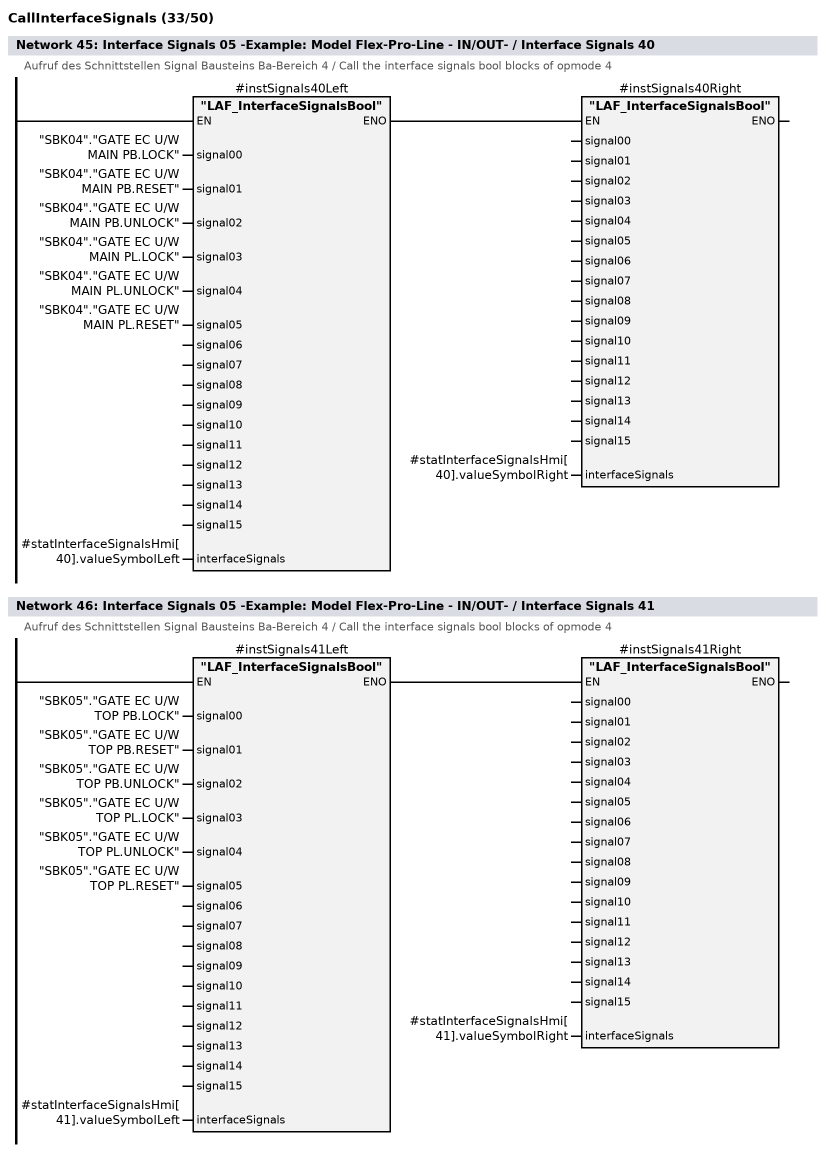
   RUNG wire#powerrail
      #instSignals40Left(signal00 := "SBK04"."GATE EC U/W MAIN PB.LOCK", signal01 := "SBK04"."GATE EC U/W MAIN PB.RESET", signal02 := "SBK04"."GATE EC U/W MAIN PB.UNLOCK", signal03 := "SBK04"."GATE EC U/W MAIN PL.LOCK", signal04 := "SBK04"."GATE EC U/W MAIN PL.UNLOCK", signal05 := "SBK04"."GATE EC U/W MAIN PL.RESET", signal06 :=, signal07 :=, signal08 :=, signal09 :=, signal10 :=, signal11 :=, signal12 :=, signal13 :=, signal14 :=, signal15 :=, interfaceSignals := #statInterfaceSignalsHmi[40].valueSymbolLeft)
      #instSignals40Right(signal00 :=, signal01 :=, signal02 :=, signal03 :=, signal04 :=, signal05 :=, signal06 :=, signal07 :=, signal08 :=, signal09 :=, signal10 :=, signal11 :=, signal12 :=, signal13 :=, signal14 :=, signal15 :=, interfaceSignals := #statInterfaceSignalsHmi[40].valueSymbolRight)
   END_RUNG
   // the same network as SCL:
   #instSignals40Left(signal00 := "SBK04"."GATE EC U/W MAIN PB.LOCK",   // "LAF_InterfaceSignalsBool"
                      signal01 := "SBK04"."GATE EC U/W MAIN PB.RESET",
                      signal02 := "SBK04"."GATE EC U/W MAIN PB.UNLOCK",
                      signal03 := "SBK04"."GATE EC U/W MAIN PL.LOCK",
                      signal04 := "SBK04"."GATE EC U/W MAIN PL.UNLOCK",
                      signal05 := "SBK04"."GATE EC U/W MAIN PL.RESET",
                      interfaceSignals := #statInterfaceSignalsHmi[40].valueSymbolLeft,
                      ENO => #_w1);
   IF #_w1 THEN
       #instSignals40Right(interfaceSignals := #statInterfaceSignalsHmi[40].valueSymbolRight);   // "LAF_InterfaceSignalsBool"
   END_IF;
END_REGION

REGION Network 46: Interface Signals 05 -Example: Model Flex-Pro-Line - IN/OUT- / Interface Signals 41
   // Aufruf des Schnittstellen Signal Bausteins Ba-Bereich 4 / Call the interface signals bool blocks of opmode 4
   RUNG wire#powerrail
      #instSignals41Left(signal00 := "SBK05"."GATE EC U/W TOP PB.LOCK", signal01 := "SBK05"."GATE EC U/W TOP PB.RESET", signal02 := "SBK05"."GATE EC U/W TOP PB.UNLOCK", signal03 := "SBK05"."GATE EC U/W TOP PL.LOCK", signal04 := "SBK05"."GATE EC U/W TOP PL.UNLOCK", signal05 := "SBK05"."GATE EC U/W TOP PL.RESET", signal06 :=, signal07 :=, signal08 :=, signal09 :=, signal10 :=, signal11 :=, signal12 :=, signal13 :=, signal14 :=, signal15 :=, interfaceSignals := #statInterfaceSignalsHmi[41].valueSymbolLeft)
      #instSignals41Right(signal00 :=, signal01 :=, signal02 :=, signal03 :=, signal04 :=, signal05 :=, signal06 :=, signal07 :=, signal08 :=, signal09 :=, signal10 :=, signal11 :=, signal12 :=, signal13 :=, signal14 :=, signal15 :=, interfaceSignals := #statInterfaceSignalsHmi[41].valueSymbolRight)
   END_RUNG
   // the same network as SCL:
   #instSignals41Left(signal00 := "SBK05"."GATE EC U/W TOP PB.LOCK",   // "LAF_InterfaceSignalsBool"
                      signal01 := "SBK05"."GATE EC U/W TOP PB.RESET",
                      signal02 := "SBK05"."GATE EC U/W TOP PB.UNLOCK",
                      signal03 := "SBK05"."GATE EC U/W TOP PL.LOCK",
                      signal04 := "SBK05"."GATE EC U/W TOP PL.UNLOCK",
                      signal05 := "SBK05"."GATE EC U/W TOP PL.RESET",
                      interfaceSignals := #statInterfaceSignalsHmi[41].valueSymbolLeft,
                      ENO => #_w1);
   IF #_w1 THEN
       #instSignals41Right(interfaceSignals := #statInterfaceSignalsHmi[41].valueSymbolRight);   // "LAF_InterfaceSignalsBool"
   END_IF;
END_REGION

REGION Network 47: Interface Signals 05 -Example: Model Flex-Pro-Line - IN/OUT- / Interface Signals 42
   // Aufruf des Schnittstellen Signal Bausteins Ba-Bereich 4 / Call the interface signals bool blocks of opmode 4
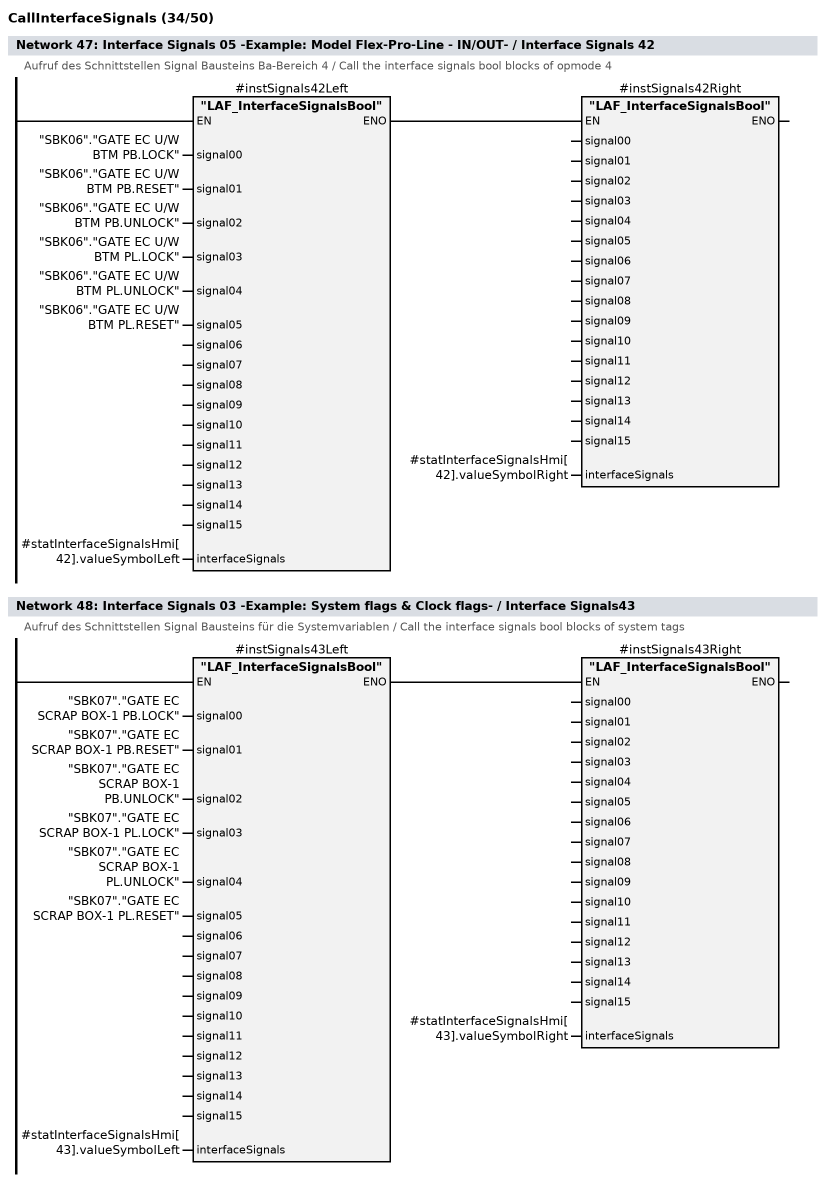
   RUNG wire#powerrail
      #instSignals42Left(signal00 := "SBK06"."GATE EC U/W BTM PB.LOCK", signal01 := "SBK06"."GATE EC U/W BTM PB.RESET", signal02 := "SBK06"."GATE EC U/W BTM PB.UNLOCK", signal03 := "SBK06"."GATE EC U/W BTM PL.LOCK", signal04 := "SBK06"."GATE EC U/W BTM PL.UNLOCK", signal05 := "SBK06"."GATE EC U/W BTM PL.RESET", signal06 :=, signal07 :=, signal08 :=, signal09 :=, signal10 :=, signal11 :=, signal12 :=, signal13 :=, signal14 :=, signal15 :=, interfaceSignals := #statInterfaceSignalsHmi[42].valueSymbolLeft)
      #instSignals42Right(signal00 :=, signal01 :=, signal02 :=, signal03 :=, signal04 :=, signal05 :=, signal06 :=, signal07 :=, signal08 :=, signal09 :=, signal10 :=, signal11 :=, signal12 :=, signal13 :=, signal14 :=, signal15 :=, interfaceSignals := #statInterfaceSignalsHmi[42].valueSymbolRight)
   END_RUNG
   // the same network as SCL:
   #instSignals42Left(signal00 := "SBK06"."GATE EC U/W BTM PB.LOCK",   // "LAF_InterfaceSignalsBool"
                      signal01 := "SBK06"."GATE EC U/W BTM PB.RESET",
                      signal02 := "SBK06"."GATE EC U/W BTM PB.UNLOCK",
                      signal03 := "SBK06"."GATE EC U/W BTM PL.LOCK",
                      signal04 := "SBK06"."GATE EC U/W BTM PL.UNLOCK",
                      signal05 := "SBK06"."GATE EC U/W BTM PL.RESET",
                      interfaceSignals := #statInterfaceSignalsHmi[42].valueSymbolLeft,
                      ENO => #_w1);
   IF #_w1 THEN
       #instSignals42Right(interfaceSignals := #statInterfaceSignalsHmi[42].valueSymbolRight);   // "LAF_InterfaceSignalsBool"
   END_IF;
END_REGION

REGION Network 48: Interface Signals 03 -Example: System flags & Clock flags- / Interface Signals43
   // Aufruf des Schnittstellen Signal Bausteins für die Systemvariablen / Call the interface signals bool blocks of system tags
   RUNG wire#powerrail
      #instSignals43Left(signal00 := "SBK07"."GATE EC SCRAP BOX-1 PB.LOCK", signal01 := "SBK07"."GATE EC SCRAP BOX-1 PB.RESET", signal02 := "SBK07"."GATE EC SCRAP BOX-1 PB.UNLOCK", signal03 := "SBK07"."GATE EC SCRAP BOX-1 PL.LOCK", signal04 := "SBK07"."GATE EC SCRAP BOX-1 PL.UNLOCK", signal05 := "SBK07"."GATE EC SCRAP BOX-1 PL.RESET", signal06 :=, signal07 :=, signal08 :=, signal09 :=, signal10 :=, signal11 :=, signal12 :=, signal13 :=, signal14 :=, signal15 :=, interfaceSignals := #statInterfaceSignalsHmi[43].valueSymbolLeft)
      #instSignals43Right(signal00 :=, signal01 :=, signal02 :=, signal03 :=, signal04 :=, signal05 :=, signal06 :=, signal07 :=, signal08 :=, signal09 :=, signal10 :=, signal11 :=, signal12 :=, signal13 :=, signal14 :=, signal15 :=, interfaceSignals := #statInterfaceSignalsHmi[43].valueSymbolRight)
   END_RUNG
   // the same network as SCL:
   #instSignals43Left(signal00 := "SBK07"."GATE EC SCRAP BOX-1 PB.LOCK",   // "LAF_InterfaceSignalsBool"
                      signal01 := "SBK07"."GATE EC SCRAP BOX-1 PB.RESET",
                      signal02 := "SBK07"."GATE EC SCRAP BOX-1 PB.UNLOCK",
                      signal03 := "SBK07"."GATE EC SCRAP BOX-1 PL.LOCK",
                      signal04 := "SBK07"."GATE EC SCRAP BOX-1 PL.UNLOCK",
                      signal05 := "SBK07"."GATE EC SCRAP BOX-1 PL.RESET",
                      interfaceSignals := #statInterfaceSignalsHmi[43].valueSymbolLeft,
                      ENO => #_w1);
   IF #_w1 THEN
       #instSignals43Right(interfaceSignals := #statInterfaceSignalsHmi[43].valueSymbolRight);   // "LAF_InterfaceSignalsBool"
   END_IF;
END_REGION

REGION Network 49: Interface Signals 04 -Example: Model Flex-Pro-Line - IN/OUT- / Interface Signals 44
   // Aufruf des Schnittstellen Signal Bausteins Ba-Bereich 4 / Call the interface signals bool blocks of opmode 4
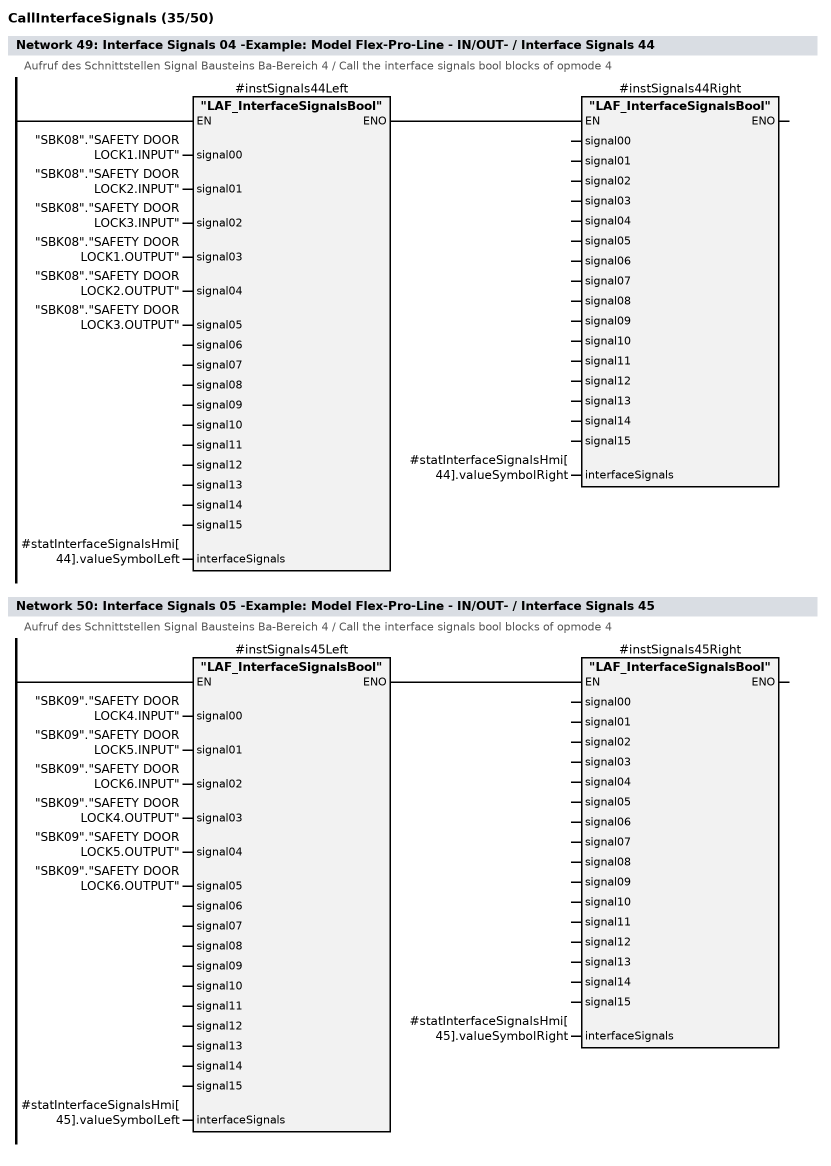
   RUNG wire#powerrail
      #instSignals44Left(signal00 := "SBK08"."SAFETY DOOR LOCK1.INPUT", signal01 := "SBK08"."SAFETY DOOR LOCK2.INPUT", signal02 := "SBK08"."SAFETY DOOR LOCK3.INPUT", signal03 := "SBK08"."SAFETY DOOR LOCK1.OUTPUT", signal04 := "SBK08"."SAFETY DOOR LOCK2.OUTPUT", signal05 := "SBK08"."SAFETY DOOR LOCK3.OUTPUT", signal06 :=, signal07 :=, signal08 :=, signal09 :=, signal10 :=, signal11 :=, signal12 :=, signal13 :=, signal14 :=, signal15 :=, interfaceSignals := #statInterfaceSignalsHmi[44].valueSymbolLeft)
      #instSignals44Right(signal00 :=, signal01 :=, signal02 :=, signal03 :=, signal04 :=, signal05 :=, signal06 :=, signal07 :=, signal08 :=, signal09 :=, signal10 :=, signal11 :=, signal12 :=, signal13 :=, signal14 :=, signal15 :=, interfaceSignals := #statInterfaceSignalsHmi[44].valueSymbolRight)
   END_RUNG
   // the same network as SCL:
   #instSignals44Left(signal00 := "SBK08"."SAFETY DOOR LOCK1.INPUT",   // "LAF_InterfaceSignalsBool"
                      signal01 := "SBK08"."SAFETY DOOR LOCK2.INPUT",
                      signal02 := "SBK08"."SAFETY DOOR LOCK3.INPUT",
                      signal03 := "SBK08"."SAFETY DOOR LOCK1.OUTPUT",
                      signal04 := "SBK08"."SAFETY DOOR LOCK2.OUTPUT",
                      signal05 := "SBK08"."SAFETY DOOR LOCK3.OUTPUT",
                      interfaceSignals := #statInterfaceSignalsHmi[44].valueSymbolLeft,
                      ENO => #_w1);
   IF #_w1 THEN
       #instSignals44Right(interfaceSignals := #statInterfaceSignalsHmi[44].valueSymbolRight);   // "LAF_InterfaceSignalsBool"
   END_IF;
END_REGION

REGION Network 50: Interface Signals 05 -Example: Model Flex-Pro-Line - IN/OUT- / Interface Signals 45
   // Aufruf des Schnittstellen Signal Bausteins Ba-Bereich 4 / Call the interface signals bool blocks of opmode 4
   RUNG wire#powerrail
      #instSignals45Left(signal00 := "SBK09"."SAFETY DOOR LOCK4.INPUT", signal01 := "SBK09"."SAFETY DOOR LOCK5.INPUT", signal02 := "SBK09"."SAFETY DOOR LOCK6.INPUT", signal03 := "SBK09"."SAFETY DOOR LOCK4.OUTPUT", signal04 := "SBK09"."SAFETY DOOR LOCK5.OUTPUT", signal05 := "SBK09"."SAFETY DOOR LOCK6.OUTPUT", signal06 :=, signal07 :=, signal08 :=, signal09 :=, signal10 :=, signal11 :=, signal12 :=, signal13 :=, signal14 :=, signal15 :=, interfaceSignals := #statInterfaceSignalsHmi[45].valueSymbolLeft)
      #instSignals45Right(signal00 :=, signal01 :=, signal02 :=, signal03 :=, signal04 :=, signal05 :=, signal06 :=, signal07 :=, signal08 :=, signal09 :=, signal10 :=, signal11 :=, signal12 :=, signal13 :=, signal14 :=, signal15 :=, interfaceSignals := #statInterfaceSignalsHmi[45].valueSymbolRight)
   END_RUNG
   // the same network as SCL:
   #instSignals45Left(signal00 := "SBK09"."SAFETY DOOR LOCK4.INPUT",   // "LAF_InterfaceSignalsBool"
                      signal01 := "SBK09"."SAFETY DOOR LOCK5.INPUT",
                      signal02 := "SBK09"."SAFETY DOOR LOCK6.INPUT",
                      signal03 := "SBK09"."SAFETY DOOR LOCK4.OUTPUT",
                      signal04 := "SBK09"."SAFETY DOOR LOCK5.OUTPUT",
                      signal05 := "SBK09"."SAFETY DOOR LOCK6.OUTPUT",
                      interfaceSignals := #statInterfaceSignalsHmi[45].valueSymbolLeft,
                      ENO => #_w1);
   IF #_w1 THEN
       #instSignals45Right(interfaceSignals := #statInterfaceSignalsHmi[45].valueSymbolRight);   // "LAF_InterfaceSignalsBool"
   END_IF;
END_REGION

REGION Network 51: Interface Signals 05 -Example: Model Flex-Pro-Line - IN/OUT- / Interface Signals 46
   // Aufruf des Schnittstellen Signal Bausteins Ba-Bereich 4 / Call the interface signals bool blocks of opmode 4
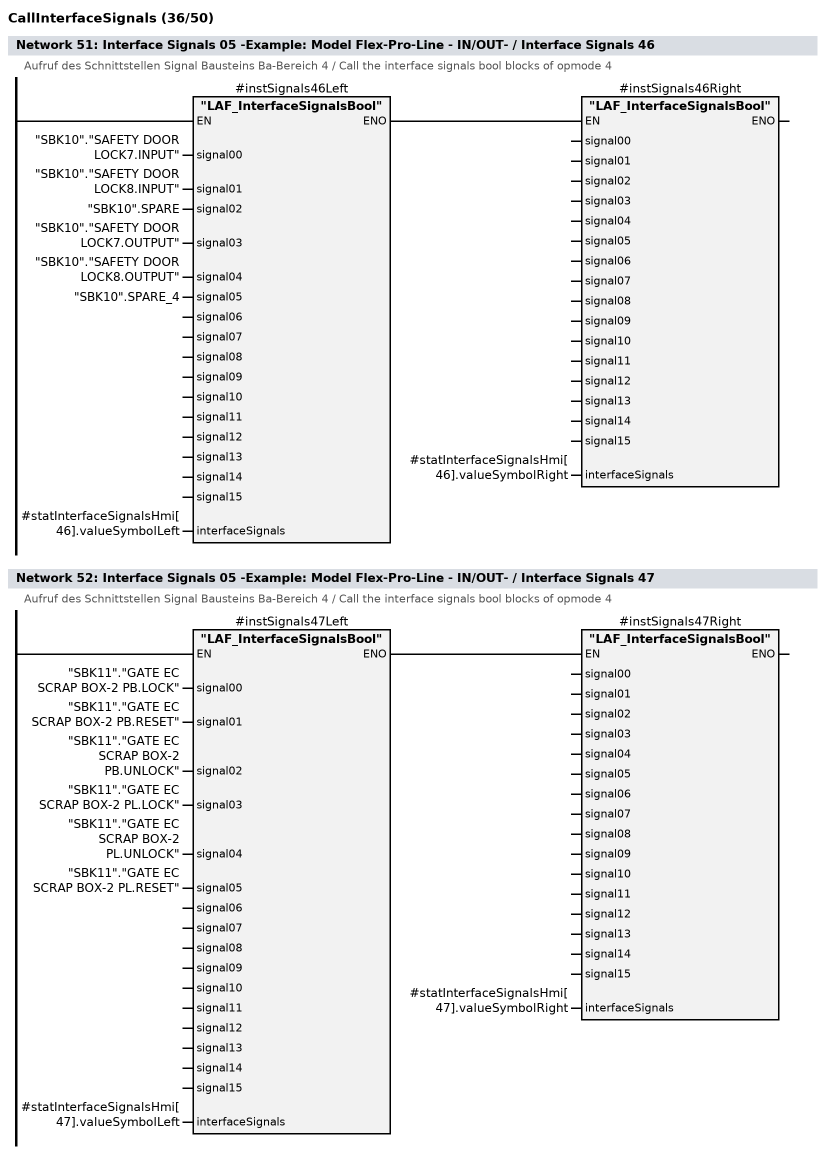
   RUNG wire#powerrail
      #instSignals46Left(signal00 := "SBK10"."SAFETY DOOR LOCK7.INPUT", signal01 := "SBK10"."SAFETY DOOR LOCK8.INPUT", signal02 := "SBK10".SPARE, signal03 := "SBK10"."SAFETY DOOR LOCK7.OUTPUT", signal04 := "SBK10"."SAFETY DOOR LOCK8.OUTPUT", signal05 := "SBK10".SPARE_4, signal06 :=, signal07 :=, signal08 :=, signal09 :=, signal10 :=, signal11 :=, signal12 :=, signal13 :=, signal14 :=, signal15 :=, interfaceSignals := #statInterfaceSignalsHmi[46].valueSymbolLeft)
      #instSignals46Right(signal00 :=, signal01 :=, signal02 :=, signal03 :=, signal04 :=, signal05 :=, signal06 :=, signal07 :=, signal08 :=, signal09 :=, signal10 :=, signal11 :=, signal12 :=, signal13 :=, signal14 :=, signal15 :=, interfaceSignals := #statInterfaceSignalsHmi[46].valueSymbolRight)
   END_RUNG
   // the same network as SCL:
   #instSignals46Left(signal00 := "SBK10"."SAFETY DOOR LOCK7.INPUT",   // "LAF_InterfaceSignalsBool"
                      signal01 := "SBK10"."SAFETY DOOR LOCK8.INPUT",
                      signal02 := "SBK10".SPARE,
                      signal03 := "SBK10"."SAFETY DOOR LOCK7.OUTPUT",
                      signal04 := "SBK10"."SAFETY DOOR LOCK8.OUTPUT",
                      signal05 := "SBK10".SPARE_4,
                      interfaceSignals := #statInterfaceSignalsHmi[46].valueSymbolLeft,
                      ENO => #_w1);
   IF #_w1 THEN
       #instSignals46Right(interfaceSignals := #statInterfaceSignalsHmi[46].valueSymbolRight);   // "LAF_InterfaceSignalsBool"
   END_IF;
END_REGION

REGION Network 52: Interface Signals 05 -Example: Model Flex-Pro-Line - IN/OUT- / Interface Signals 47
   // Aufruf des Schnittstellen Signal Bausteins Ba-Bereich 4 / Call the interface signals bool blocks of opmode 4
   RUNG wire#powerrail
      #instSignals47Left(signal00 := "SBK11"."GATE EC SCRAP BOX-2 PB.LOCK", signal01 := "SBK11"."GATE EC SCRAP BOX-2 PB.RESET", signal02 := "SBK11"."GATE EC SCRAP BOX-2 PB.UNLOCK", signal03 := "SBK11"."GATE EC SCRAP BOX-2 PL.LOCK", signal04 := "SBK11"."GATE EC SCRAP BOX-2 PL.UNLOCK", signal05 := "SBK11"."GATE EC SCRAP BOX-2 PL.RESET", signal06 :=, signal07 :=, signal08 :=, signal09 :=, signal10 :=, signal11 :=, signal12 :=, signal13 :=, signal14 :=, signal15 :=, interfaceSignals := #statInterfaceSignalsHmi[47].valueSymbolLeft)
      #instSignals47Right(signal00 :=, signal01 :=, signal02 :=, signal03 :=, signal04 :=, signal05 :=, signal06 :=, signal07 :=, signal08 :=, signal09 :=, signal10 :=, signal11 :=, signal12 :=, signal13 :=, signal14 :=, signal15 :=, interfaceSignals := #statInterfaceSignalsHmi[47].valueSymbolRight)
   END_RUNG
   // the same network as SCL:
   #instSignals47Left(signal00 := "SBK11"."GATE EC SCRAP BOX-2 PB.LOCK",   // "LAF_InterfaceSignalsBool"
                      signal01 := "SBK11"."GATE EC SCRAP BOX-2 PB.RESET",
                      signal02 := "SBK11"."GATE EC SCRAP BOX-2 PB.UNLOCK",
                      signal03 := "SBK11"."GATE EC SCRAP BOX-2 PL.LOCK",
                      signal04 := "SBK11"."GATE EC SCRAP BOX-2 PL.UNLOCK",
                      signal05 := "SBK11"."GATE EC SCRAP BOX-2 PL.RESET",
                      interfaceSignals := #statInterfaceSignalsHmi[47].valueSymbolLeft,
                      ENO => #_w1);
   IF #_w1 THEN
       #instSignals47Right(interfaceSignals := #statInterfaceSignalsHmi[47].valueSymbolRight);   // "LAF_InterfaceSignalsBool"
   END_IF;
END_REGION

REGION Network 53: Interface Signals 05 -Example: Model Flex-Pro-Line - IN/OUT- / Interface Signals 48
   // Aufruf des Schnittstellen Signal Bausteins Ba-Bereich 4 / Call the interface signals bool blocks of opmode 4
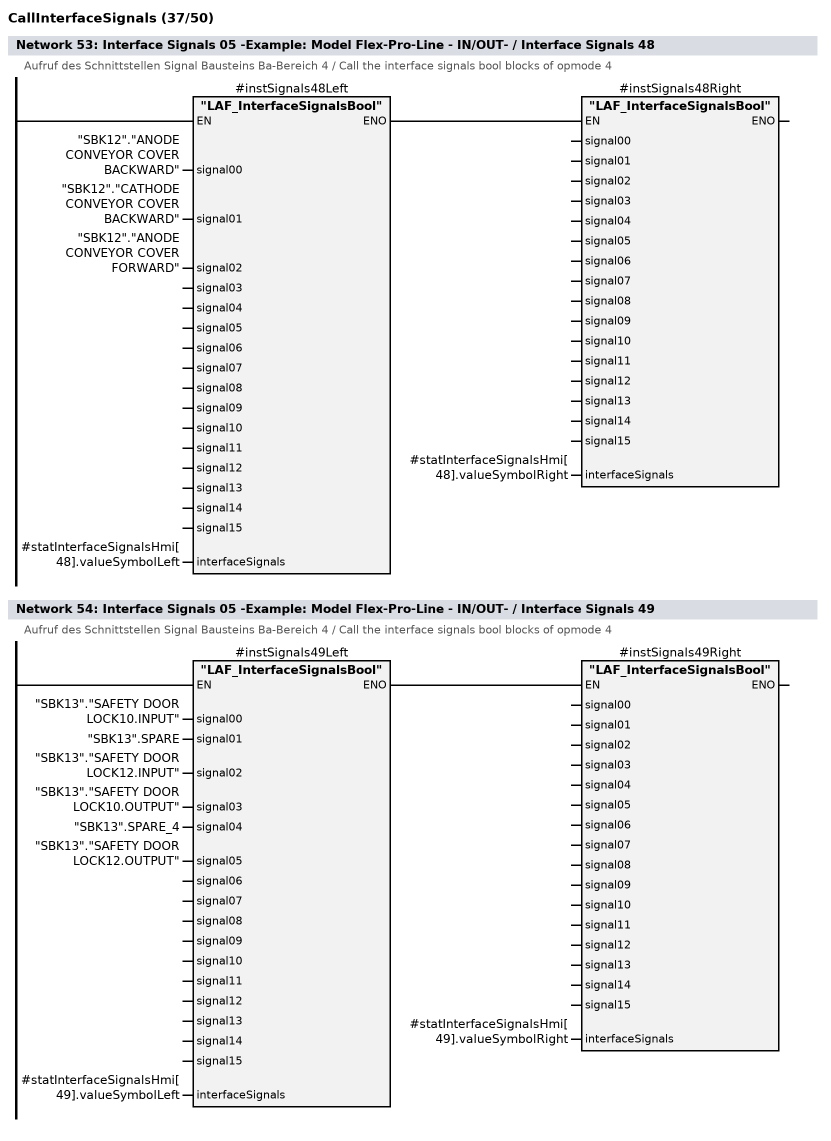
   RUNG wire#powerrail
      #instSignals48Left(signal00 := "SBK12"."ANODE CONVEYOR COVER BACKWARD", signal01 := "SBK12"."CATHODE CONVEYOR COVER BACKWARD", signal02 := "SBK12"."ANODE CONVEYOR COVER FORWARD", signal03 :=, signal04 :=, signal05 :=, signal06 :=, signal07 :=, signal08 :=, signal09 :=, signal10 :=, signal11 :=, signal12 :=, signal13 :=, signal14 :=, signal15 :=, interfaceSignals := #statInterfaceSignalsHmi[48].valueSymbolLeft)
      #instSignals48Right(signal00 :=, signal01 :=, signal02 :=, signal03 :=, signal04 :=, signal05 :=, signal06 :=, signal07 :=, signal08 :=, signal09 :=, signal10 :=, signal11 :=, signal12 :=, signal13 :=, signal14 :=, signal15 :=, interfaceSignals := #statInterfaceSignalsHmi[48].valueSymbolRight)
   END_RUNG
   // the same network as SCL:
   #instSignals48Left(signal00 := "SBK12"."ANODE CONVEYOR COVER BACKWARD",   // "LAF_InterfaceSignalsBool"
                      signal01 := "SBK12"."CATHODE CONVEYOR COVER BACKWARD",
                      signal02 := "SBK12"."ANODE CONVEYOR COVER FORWARD",
                      interfaceSignals := #statInterfaceSignalsHmi[48].valueSymbolLeft,
                      ENO => #_w1);
   IF #_w1 THEN
       #instSignals48Right(interfaceSignals := #statInterfaceSignalsHmi[48].valueSymbolRight);   // "LAF_InterfaceSignalsBool"
   END_IF;
END_REGION

REGION Network 54: Interface Signals 05 -Example: Model Flex-Pro-Line - IN/OUT- / Interface Signals 49
   // Aufruf des Schnittstellen Signal Bausteins Ba-Bereich 4 / Call the interface signals bool blocks of opmode 4
   RUNG wire#powerrail
      #instSignals49Left(signal00 := "SBK13"."SAFETY DOOR LOCK10.INPUT", signal01 := "SBK13".SPARE, signal02 := "SBK13"."SAFETY DOOR LOCK12.INPUT", signal03 := "SBK13"."SAFETY DOOR LOCK10.OUTPUT", signal04 := "SBK13".SPARE_4, signal05 := "SBK13"."SAFETY DOOR LOCK12.OUTPUT", signal06 :=, signal07 :=, signal08 :=, signal09 :=, signal10 :=, signal11 :=, signal12 :=, signal13 :=, signal14 :=, signal15 :=, interfaceSignals := #statInterfaceSignalsHmi[49].valueSymbolLeft)
      #instSignals49Right(signal00 :=, signal01 :=, signal02 :=, signal03 :=, signal04 :=, signal05 :=, signal06 :=, signal07 :=, signal08 :=, signal09 :=, signal10 :=, signal11 :=, signal12 :=, signal13 :=, signal14 :=, signal15 :=, interfaceSignals := #statInterfaceSignalsHmi[49].valueSymbolRight)
   END_RUNG
   // the same network as SCL:
   #instSignals49Left(signal00 := "SBK13"."SAFETY DOOR LOCK10.INPUT",   // "LAF_InterfaceSignalsBool"
                      signal01 := "SBK13".SPARE,
                      signal02 := "SBK13"."SAFETY DOOR LOCK12.INPUT",
                      signal03 := "SBK13"."SAFETY DOOR LOCK10.OUTPUT",
                      signal04 := "SBK13".SPARE_4,
                      signal05 := "SBK13"."SAFETY DOOR LOCK12.OUTPUT",
                      interfaceSignals := #statInterfaceSignalsHmi[49].valueSymbolLeft,
                      ENO => #_w1);
   IF #_w1 THEN
       #instSignals49Right(interfaceSignals := #statInterfaceSignalsHmi[49].valueSymbolRight);   // "LAF_InterfaceSignalsBool"
   END_IF;
END_REGION

REGION Network 55: Interface Signals 05 -Example: Model Flex-Pro-Line - IN/OUT- / Interface Signals 50
   // Aufruf des Schnittstellen Signal Bausteins Ba-Bereich 4 / Call the interface signals bool blocks of opmode 4
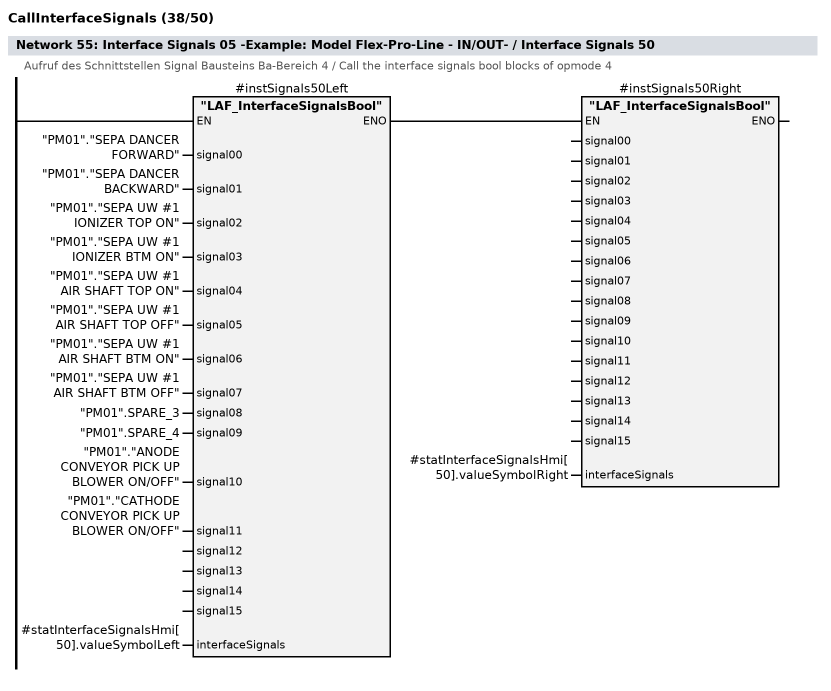
   RUNG wire#powerrail
      #instSignals50Left(signal00 := "PM01"."SEPA DANCER FORWARD", signal01 := "PM01"."SEPA DANCER BACKWARD", signal02 := "PM01"."SEPA UW #1 IONIZER TOP ON", signal03 := "PM01"."SEPA UW #1 IONIZER BTM ON", signal04 := "PM01"."SEPA UW #1 AIR SHAFT TOP ON", signal05 := "PM01"."SEPA UW #1 AIR SHAFT TOP OFF", signal06 := "PM01"."SEPA UW #1 AIR SHAFT BTM ON", signal07 := "PM01"."SEPA UW #1 AIR SHAFT BTM OFF", signal08 := "PM01".SPARE_3, signal09 := "PM01".SPARE_4, signal10 := "PM01"."ANODE CONVEYOR PICK UP BLOWER ON/OFF", signal11 := "PM01"."CATHODE CONVEYOR PICK UP BLOWER ON/OFF", signal12 :=, signal13 :=, signal14 :=, signal15 :=, interfaceSignals := #statInterfaceSignalsHmi[50].valueSymbolLeft)
      #instSignals50Right(signal00 :=, signal01 :=, signal02 :=, signal03 :=, signal04 :=, signal05 :=, signal06 :=, signal07 :=, signal08 :=, signal09 :=, signal10 :=, signal11 :=, signal12 :=, signal13 :=, signal14 :=, signal15 :=, interfaceSignals := #statInterfaceSignalsHmi[50].valueSymbolRight)
   END_RUNG
   // the same network as SCL:
   #instSignals50Left(signal00 := "PM01"."SEPA DANCER FORWARD",   // "LAF_InterfaceSignalsBool"
                      signal01 := "PM01"."SEPA DANCER BACKWARD",
                      signal02 := "PM01"."SEPA UW #1 IONIZER TOP ON",
                      signal03 := "PM01"."SEPA UW #1 IONIZER BTM ON",
                      signal04 := "PM01"."SEPA UW #1 AIR SHAFT TOP ON",
                      signal05 := "PM01"."SEPA UW #1 AIR SHAFT TOP OFF",
                      signal06 := "PM01"."SEPA UW #1 AIR SHAFT BTM ON",
                      signal07 := "PM01"."SEPA UW #1 AIR SHAFT BTM OFF",
                      signal08 := "PM01".SPARE_3,
                      signal09 := "PM01".SPARE_4,
                      signal10 := "PM01"."ANODE CONVEYOR PICK UP BLOWER ON/OFF",
                      signal11 := "PM01"."CATHODE CONVEYOR PICK UP BLOWER ON/OFF",
                      interfaceSignals := #statInterfaceSignalsHmi[50].valueSymbolLeft,
                      ENO => #_w1);
   IF #_w1 THEN
       #instSignals50Right(interfaceSignals := #statInterfaceSignalsHmi[50].valueSymbolRight);   // "LAF_InterfaceSignalsBool"
   END_IF;
END_REGION

REGION Network 56: Interface Signals 05 -Example: Model Flex-Pro-Line - IN/OUT- / Interface Signals 51
   // Aufruf des Schnittstellen Signal Bausteins Ba-Bereich 4 / Call the interface signals bool blocks of opmode 4
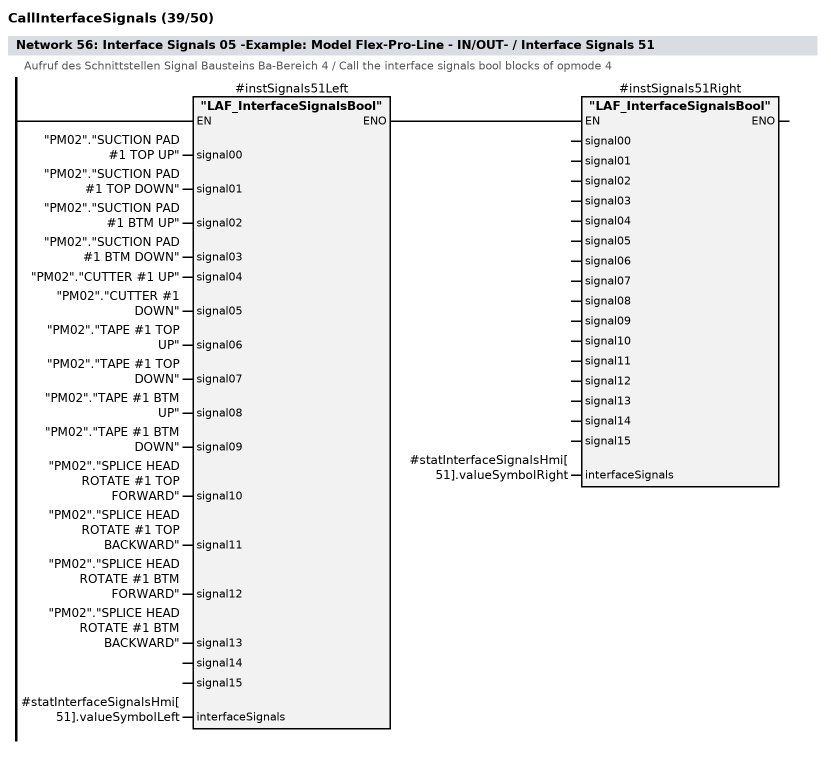
   RUNG wire#powerrail
      #instSignals51Left(signal00 := "PM02"."SUCTION PAD #1 TOP UP", signal01 := "PM02"."SUCTION PAD #1 TOP DOWN", signal02 := "PM02"."SUCTION PAD #1 BTM UP", signal03 := "PM02"."SUCTION PAD #1 BTM DOWN", signal04 := "PM02"."CUTTER #1 UP", signal05 := "PM02"."CUTTER #1 DOWN", signal06 := "PM02"."TAPE #1 TOP UP", signal07 := "PM02"."TAPE #1 TOP DOWN", signal08 := "PM02"."TAPE #1 BTM UP", signal09 := "PM02"."TAPE #1 BTM DOWN", signal10 := "PM02"."SPLICE HEAD ROTATE #1 TOP FORWARD", signal11 := "PM02"."SPLICE HEAD ROTATE #1 TOP BACKWARD", signal12 := "PM02"."SPLICE HEAD ROTATE #1 BTM FORWARD", signal13 := "PM02"."SPLICE HEAD ROTATE #1 BTM BACKWARD", signal14 :=, signal15 :=, interfaceSignals := #statInterfaceSignalsHmi[51].valueSymbolLeft)
      #instSignals51Right(signal00 :=, signal01 :=, signal02 :=, signal03 :=, signal04 :=, signal05 :=, signal06 :=, signal07 :=, signal08 :=, signal09 :=, signal10 :=, signal11 :=, signal12 :=, signal13 :=, signal14 :=, signal15 :=, interfaceSignals := #statInterfaceSignalsHmi[51].valueSymbolRight)
   END_RUNG
   // the same network as SCL:
   #instSignals51Left(signal00 := "PM02"."SUCTION PAD #1 TOP UP",   // "LAF_InterfaceSignalsBool"
                      signal01 := "PM02"."SUCTION PAD #1 TOP DOWN",
                      signal02 := "PM02"."SUCTION PAD #1 BTM UP",
                      signal03 := "PM02"."SUCTION PAD #1 BTM DOWN",
                      signal04 := "PM02"."CUTTER #1 UP",
                      signal05 := "PM02"."CUTTER #1 DOWN",
                      signal06 := "PM02"."TAPE #1 TOP UP",
                      signal07 := "PM02"."TAPE #1 TOP DOWN",
                      signal08 := "PM02"."TAPE #1 BTM UP",
                      signal09 := "PM02"."TAPE #1 BTM DOWN",
                      signal10 := "PM02"."SPLICE HEAD ROTATE #1 TOP FORWARD",
                      signal11 := "PM02"."SPLICE HEAD ROTATE #1 TOP BACKWARD",
                      signal12 := "PM02"."SPLICE HEAD ROTATE #1 BTM FORWARD",
                      signal13 := "PM02"."SPLICE HEAD ROTATE #1 BTM BACKWARD",
                      interfaceSignals := #statInterfaceSignalsHmi[51].valueSymbolLeft,
                      ENO => #_w1);
   IF #_w1 THEN
       #instSignals51Right(interfaceSignals := #statInterfaceSignalsHmi[51].valueSymbolRight);   // "LAF_InterfaceSignalsBool"
   END_IF;
END_REGION

REGION Network 57: Interface Signals 05 -Example: Model Flex-Pro-Line - IN/OUT- / Interface Signals 52
   // Aufruf des Schnittstellen Signal Bausteins Ba-Bereich 4 / Call the interface signals bool blocks of opmode 4
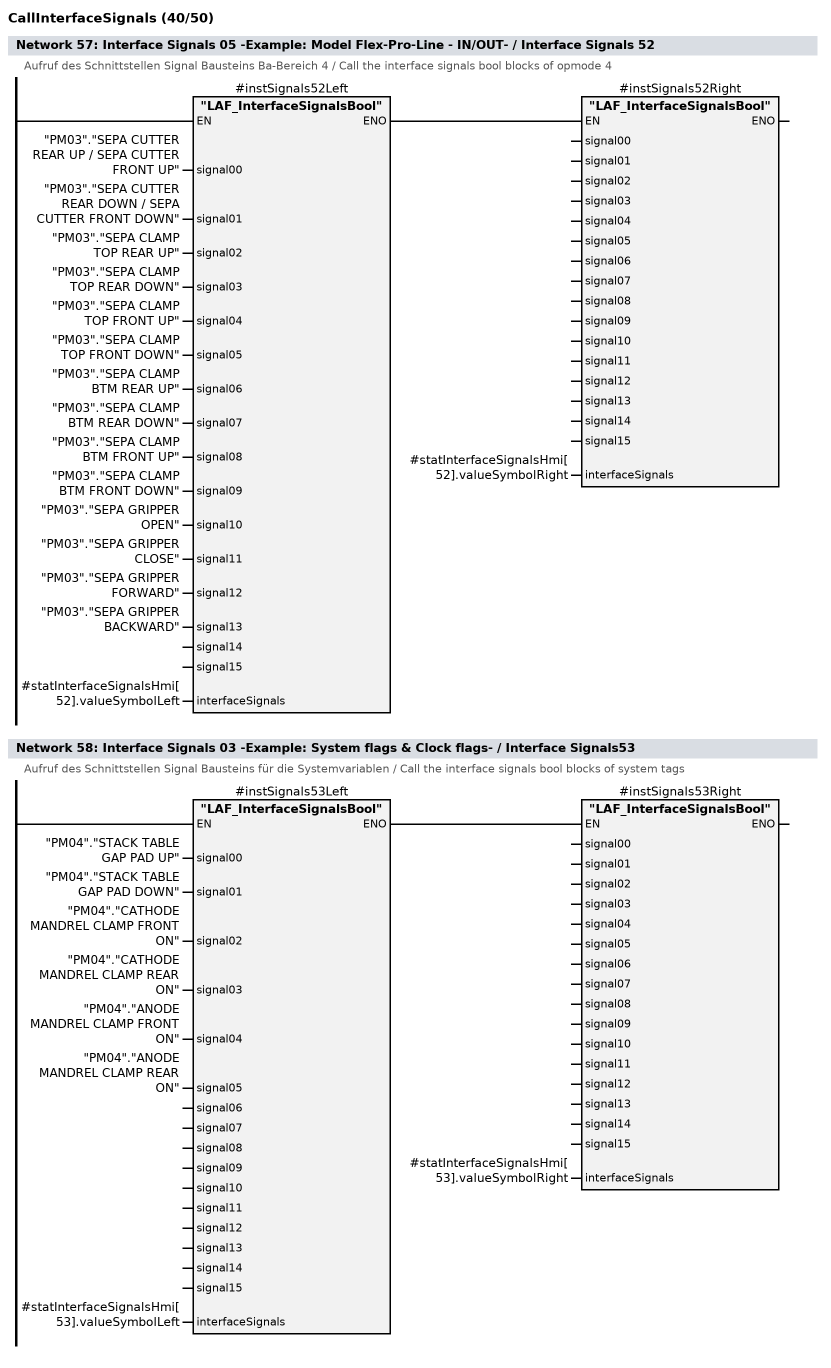
   RUNG wire#powerrail
      #instSignals52Left(signal00 := "PM03"."SEPA CUTTER REAR UP / SEPA CUTTER FRONT UP", signal01 := "PM03"."SEPA CUTTER REAR DOWN / SEPA CUTTER FRONT DOWN", signal02 := "PM03"."SEPA CLAMP TOP REAR UP", signal03 := "PM03"."SEPA CLAMP TOP REAR DOWN", signal04 := "PM03"."SEPA CLAMP TOP FRONT UP", signal05 := "PM03"."SEPA CLAMP TOP FRONT DOWN", signal06 := "PM03"."SEPA CLAMP BTM REAR UP", signal07 := "PM03"."SEPA CLAMP BTM REAR DOWN", signal08 := "PM03"."SEPA CLAMP BTM FRONT UP", signal09 := "PM03"."SEPA CLAMP BTM FRONT DOWN", signal10 := "PM03"."SEPA GRIPPER OPEN", signal11 := "PM03"."SEPA GRIPPER  CLOSE", signal12 := "PM03"."SEPA GRIPPER FORWARD", signal13 := "PM03"."SEPA GRIPPER BACKWARD", signal14 :=, signal15 :=, interfaceSignals := #statInterfaceSignalsHmi[52].valueSymbolLeft)
      #instSignals52Right(signal00 :=, signal01 :=, signal02 :=, signal03 :=, signal04 :=, signal05 :=, signal06 :=, signal07 :=, signal08 :=, signal09 :=, signal10 :=, signal11 :=, signal12 :=, signal13 :=, signal14 :=, signal15 :=, interfaceSignals := #statInterfaceSignalsHmi[52].valueSymbolRight)
   END_RUNG
   // the same network as SCL:
   #instSignals52Left(signal00 := "PM03"."SEPA CUTTER REAR UP / SEPA CUTTER FRONT UP",   // "LAF_InterfaceSignalsBool"
                      signal01 := "PM03"."SEPA CUTTER REAR DOWN / SEPA CUTTER FRONT DOWN",
                      signal02 := "PM03"."SEPA CLAMP TOP REAR UP",
                      signal03 := "PM03"."SEPA CLAMP TOP REAR DOWN",
                      signal04 := "PM03"."SEPA CLAMP TOP FRONT UP",
                      signal05 := "PM03"."SEPA CLAMP TOP FRONT DOWN",
                      signal06 := "PM03"."SEPA CLAMP BTM REAR UP",
                      signal07 := "PM03"."SEPA CLAMP BTM REAR DOWN",
                      signal08 := "PM03"."SEPA CLAMP BTM FRONT UP",
                      signal09 := "PM03"."SEPA CLAMP BTM FRONT DOWN",
                      signal10 := "PM03"."SEPA GRIPPER OPEN",
                      signal11 := "PM03"."SEPA GRIPPER  CLOSE",
                      signal12 := "PM03"."SEPA GRIPPER FORWARD",
                      signal13 := "PM03"."SEPA GRIPPER BACKWARD",
                      interfaceSignals := #statInterfaceSignalsHmi[52].valueSymbolLeft,
                      ENO => #_w1);
   IF #_w1 THEN
       #instSignals52Right(interfaceSignals := #statInterfaceSignalsHmi[52].valueSymbolRight);   // "LAF_InterfaceSignalsBool"
   END_IF;
END_REGION

REGION Network 58: Interface Signals 03 -Example: System flags & Clock flags- / Interface Signals53
   // Aufruf des Schnittstellen Signal Bausteins für die Systemvariablen / Call the interface signals bool blocks of system tags
   RUNG wire#powerrail
      #instSignals53Left(signal00 := "PM04"."STACK TABLE GAP PAD UP", signal01 := "PM04"."STACK TABLE GAP PAD DOWN", signal02 := "PM04"."CATHODE MANDREL CLAMP FRONT ON", signal03 := "PM04"."CATHODE MANDREL CLAMP REAR ON", signal04 := "PM04"."ANODE MANDREL CLAMP FRONT ON", signal05 := "PM04"."ANODE MANDREL CLAMP REAR ON", signal06 :=, signal07 :=, signal08 :=, signal09 :=, signal10 :=, signal11 :=, signal12 :=, signal13 :=, signal14 :=, signal15 :=, interfaceSignals := #statInterfaceSignalsHmi[53].valueSymbolLeft)
      #instSignals53Right(signal00 :=, signal01 :=, signal02 :=, signal03 :=, signal04 :=, signal05 :=, signal06 :=, signal07 :=, signal08 :=, signal09 :=, signal10 :=, signal11 :=, signal12 :=, signal13 :=, signal14 :=, signal15 :=, interfaceSignals := #statInterfaceSignalsHmi[53].valueSymbolRight)
   END_RUNG
   // the same network as SCL:
   #instSignals53Left(signal00 := "PM04"."STACK TABLE GAP PAD UP",   // "LAF_InterfaceSignalsBool"
                      signal01 := "PM04"."STACK TABLE GAP PAD DOWN",
                      signal02 := "PM04"."CATHODE MANDREL CLAMP FRONT ON",
                      signal03 := "PM04"."CATHODE MANDREL CLAMP REAR ON",
                      signal04 := "PM04"."ANODE MANDREL CLAMP FRONT ON",
                      signal05 := "PM04"."ANODE MANDREL CLAMP REAR ON",
                      interfaceSignals := #statInterfaceSignalsHmi[53].valueSymbolLeft,
                      ENO => #_w1);
   IF #_w1 THEN
       #instSignals53Right(interfaceSignals := #statInterfaceSignalsHmi[53].valueSymbolRight);   // "LAF_InterfaceSignalsBool"
   END_IF;
END_REGION

REGION Network 59: Interface Signals 04 -Example: Model Flex-Pro-Line - IN/OUT- / Interface Signals 54
   // Aufruf des Schnittstellen Signal Bausteins Ba-Bereich 4 / Call the interface signals bool blocks of opmode 4
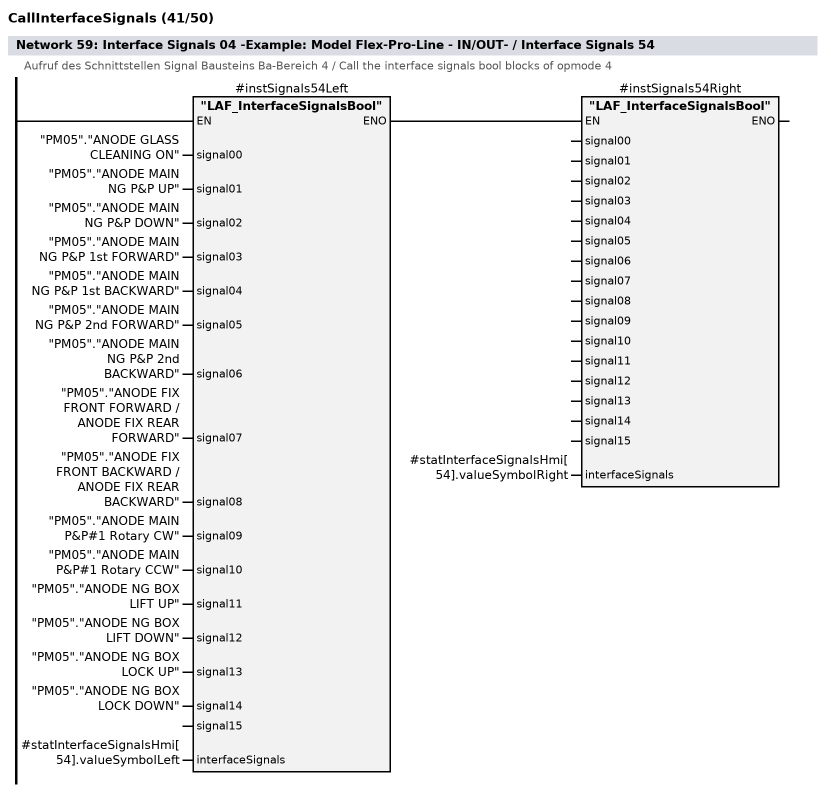
   RUNG wire#powerrail
      #instSignals54Left(signal00 := "PM05"."ANODE GLASS CLEANING ON", signal01 := "PM05"."ANODE MAIN NG P&P UP", signal02 := "PM05"."ANODE MAIN NG P&P DOWN", signal03 := "PM05"."ANODE MAIN NG P&P 1st FORWARD", signal04 := "PM05"."ANODE MAIN NG P&P 1st BACKWARD", signal05 := "PM05"."ANODE MAIN NG P&P 2nd FORWARD", signal06 := "PM05"."ANODE MAIN NG P&P 2nd BACKWARD", signal07 := "PM05"."ANODE FIX FRONT FORWARD / ANODE FIX REAR FORWARD", signal08 := "PM05"."ANODE FIX FRONT BACKWARD / ANODE FIX REAR BACKWARD", signal09 := "PM05"."ANODE MAIN P&P#1 Rotary CW", signal10 := "PM05"."ANODE MAIN P&P#1 Rotary CCW", signal11 := "PM05"."ANODE NG BOX LIFT UP", signal12 := "PM05"."ANODE NG BOX LIFT DOWN", signal13 := "PM05"."ANODE NG BOX LOCK UP", signal14 := "PM05"."ANODE NG BOX LOCK DOWN", signal15 :=, interfaceSignals := #statInterfaceSignalsHmi[54].valueSymbolLeft)
      #instSignals54Right(signal00 :=, signal01 :=, signal02 :=, signal03 :=, signal04 :=, signal05 :=, signal06 :=, signal07 :=, signal08 :=, signal09 :=, signal10 :=, signal11 :=, signal12 :=, signal13 :=, signal14 :=, signal15 :=, interfaceSignals := #statInterfaceSignalsHmi[54].valueSymbolRight)
   END_RUNG
   // the same network as SCL:
   #instSignals54Left(signal00 := "PM05"."ANODE GLASS CLEANING ON",   // "LAF_InterfaceSignalsBool"
                      signal01 := "PM05"."ANODE MAIN NG P&P UP",
                      signal02 := "PM05"."ANODE MAIN NG P&P DOWN",
                      signal03 := "PM05"."ANODE MAIN NG P&P 1st FORWARD",
                      signal04 := "PM05"."ANODE MAIN NG P&P 1st BACKWARD",
                      signal05 := "PM05"."ANODE MAIN NG P&P 2nd FORWARD",
                      signal06 := "PM05"."ANODE MAIN NG P&P 2nd BACKWARD",
                      signal07 := "PM05"."ANODE FIX FRONT FORWARD / ANODE FIX REAR FORWARD",
                      signal08 := "PM05"."ANODE FIX FRONT BACKWARD / ANODE FIX REAR BACKWARD",
                      signal09 := "PM05"."ANODE MAIN P&P#1 Rotary CW",
                      signal10 := "PM05"."ANODE MAIN P&P#1 Rotary CCW",
                      signal11 := "PM05"."ANODE NG BOX LIFT UP",
                      signal12 := "PM05"."ANODE NG BOX LIFT DOWN",
                      signal13 := "PM05"."ANODE NG BOX LOCK UP",
                      signal14 := "PM05"."ANODE NG BOX LOCK DOWN",
                      interfaceSignals := #statInterfaceSignalsHmi[54].valueSymbolLeft,
                      ENO => #_w1);
   IF #_w1 THEN
       #instSignals54Right(interfaceSignals := #statInterfaceSignalsHmi[54].valueSymbolRight);   // "LAF_InterfaceSignalsBool"
   END_IF;
END_REGION

REGION Network 60: Interface Signals 05 -Example: Model Flex-Pro-Line - IN/OUT- / Interface Signals 55
   // Aufruf des Schnittstellen Signal Bausteins Ba-Bereich 4 / Call the interface signals bool blocks of opmode 4
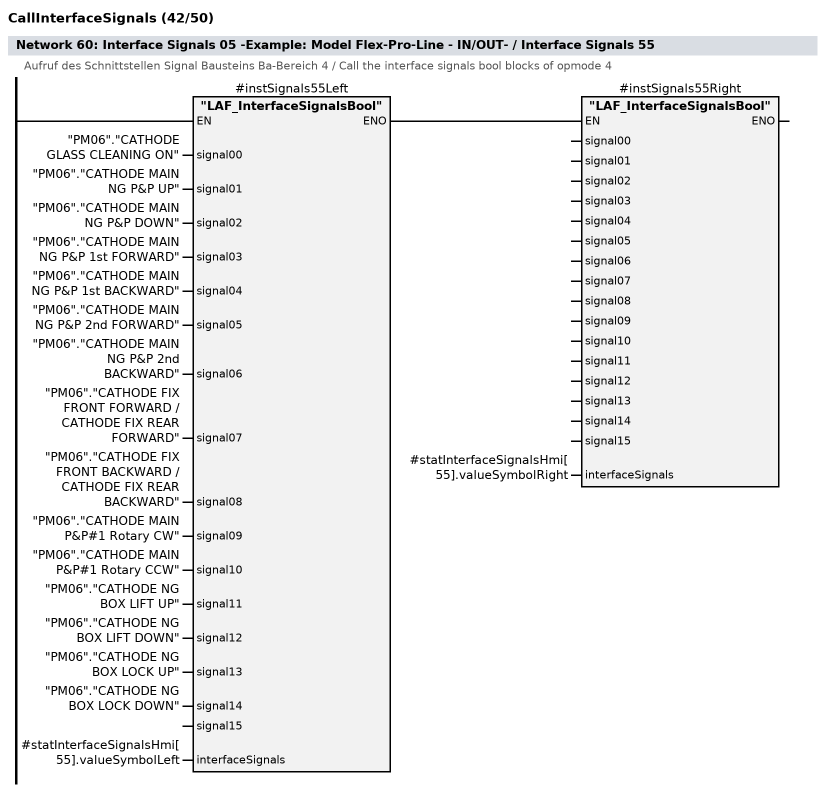
   RUNG wire#powerrail
      #instSignals55Left(signal00 := "PM06"."CATHODE GLASS CLEANING ON", signal01 := "PM06"."CATHODE MAIN NG P&P UP", signal02 := "PM06"."CATHODE MAIN NG P&P DOWN", signal03 := "PM06"."CATHODE MAIN NG P&P 1st FORWARD", signal04 := "PM06"."CATHODE MAIN NG P&P 1st BACKWARD", signal05 := "PM06"."CATHODE MAIN NG P&P 2nd FORWARD", signal06 := "PM06"."CATHODE MAIN NG P&P 2nd BACKWARD", signal07 := "PM06"."CATHODE FIX FRONT FORWARD / CATHODE FIX REAR FORWARD", signal08 := "PM06"."CATHODE FIX FRONT BACKWARD / CATHODE FIX REAR BACKWARD", signal09 := "PM06"."CATHODE MAIN P&P#1 Rotary CW", signal10 := "PM06"."CATHODE MAIN P&P#1 Rotary CCW", signal11 := "PM06"."CATHODE NG BOX LIFT UP", signal12 := "PM06"."CATHODE NG BOX LIFT DOWN", signal13 := "PM06"."CATHODE NG BOX LOCK UP", signal14 := "PM06"."CATHODE NG BOX LOCK DOWN", signal15 :=, interfaceSignals := #statInterfaceSignalsHmi[55].valueSymbolLeft)
      #instSignals55Right(signal00 :=, signal01 :=, signal02 :=, signal03 :=, signal04 :=, signal05 :=, signal06 :=, signal07 :=, signal08 :=, signal09 :=, signal10 :=, signal11 :=, signal12 :=, signal13 :=, signal14 :=, signal15 :=, interfaceSignals := #statInterfaceSignalsHmi[55].valueSymbolRight)
   END_RUNG
   // the same network as SCL:
   #instSignals55Left(signal00 := "PM06"."CATHODE GLASS CLEANING ON",   // "LAF_InterfaceSignalsBool"
                      signal01 := "PM06"."CATHODE MAIN NG P&P UP",
                      signal02 := "PM06"."CATHODE MAIN NG P&P DOWN",
                      signal03 := "PM06"."CATHODE MAIN NG P&P 1st FORWARD",
                      signal04 := "PM06"."CATHODE MAIN NG P&P 1st BACKWARD",
                      signal05 := "PM06"."CATHODE MAIN NG P&P 2nd FORWARD",
                      signal06 := "PM06"."CATHODE MAIN NG P&P 2nd BACKWARD",
                      signal07 := "PM06"."CATHODE FIX FRONT FORWARD / CATHODE FIX REAR FORWARD",
                      signal08 := "PM06"."CATHODE FIX FRONT BACKWARD / CATHODE FIX REAR BACKWARD",
                      signal09 := "PM06"."CATHODE MAIN P&P#1 Rotary CW",
                      signal10 := "PM06"."CATHODE MAIN P&P#1 Rotary CCW",
                      signal11 := "PM06"."CATHODE NG BOX LIFT UP",
                      signal12 := "PM06"."CATHODE NG BOX LIFT DOWN",
                      signal13 := "PM06"."CATHODE NG BOX LOCK UP",
                      signal14 := "PM06"."CATHODE NG BOX LOCK DOWN",
                      interfaceSignals := #statInterfaceSignalsHmi[55].valueSymbolLeft,
                      ENO => #_w1);
   IF #_w1 THEN
       #instSignals55Right(interfaceSignals := #statInterfaceSignalsHmi[55].valueSymbolRight);   // "LAF_InterfaceSignalsBool"
   END_IF;
END_REGION

REGION Network 61: Interface Signals 05 -Example: Model Flex-Pro-Line - IN/OUT- / Interface Signals 56
   // Aufruf des Schnittstellen Signal Bausteins Ba-Bereich 4 / Call the interface signals bool blocks of opmode 4
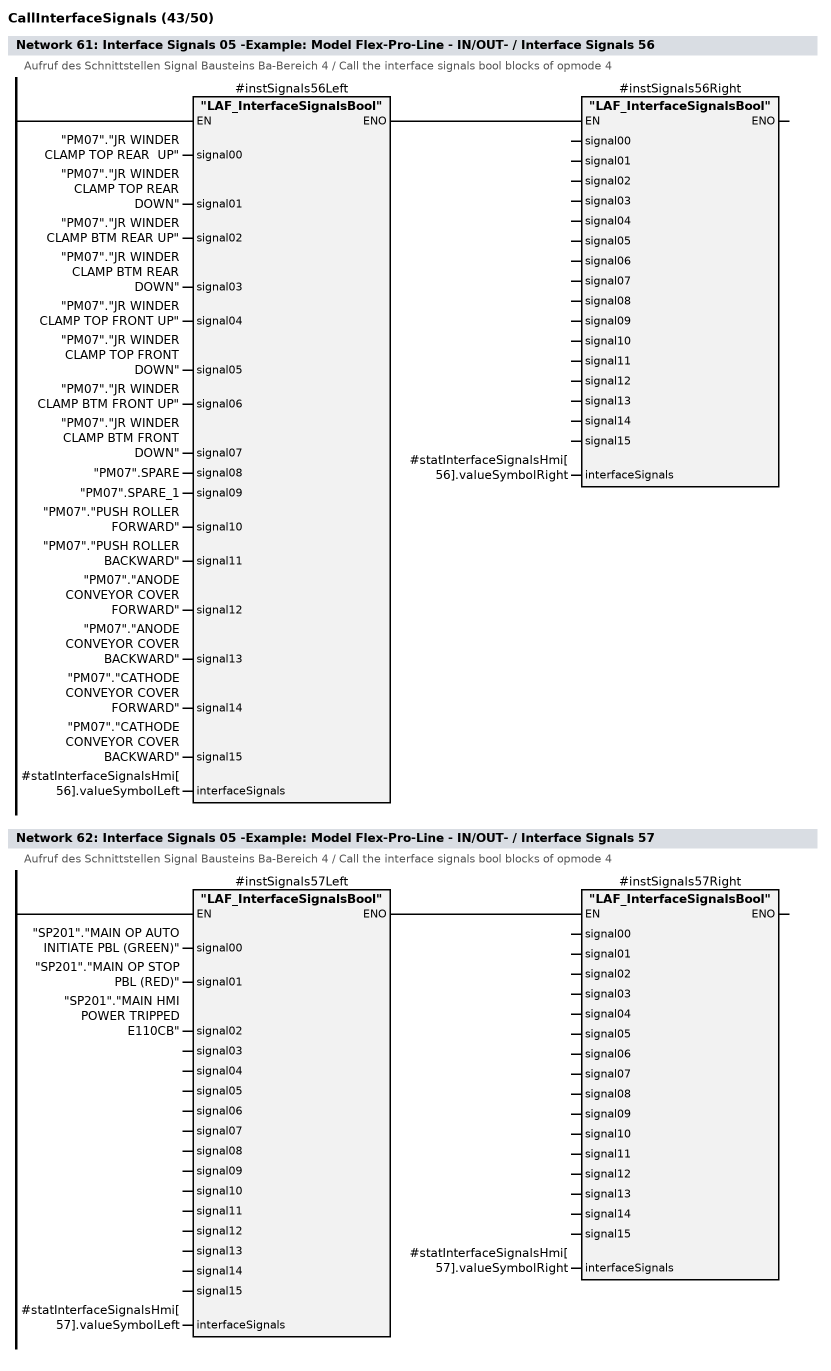
   RUNG wire#powerrail
      #instSignals56Left(signal00 := "PM07"."JR WINDER CLAMP TOP REAR  UP", signal01 := "PM07"."JR WINDER CLAMP TOP REAR  DOWN", signal02 := "PM07"."JR WINDER CLAMP BTM REAR UP", signal03 := "PM07"."JR WINDER CLAMP BTM REAR DOWN", signal04 := "PM07"."JR WINDER CLAMP TOP FRONT UP", signal05 := "PM07"."JR WINDER CLAMP TOP FRONT DOWN", signal06 := "PM07"."JR WINDER CLAMP BTM FRONT UP", signal07 := "PM07"."JR WINDER CLAMP BTM FRONT DOWN", signal08 := "PM07".SPARE, signal09 := "PM07".SPARE_1, signal10 := "PM07"."PUSH ROLLER FORWARD", signal11 := "PM07"."PUSH ROLLER BACKWARD", signal12 := "PM07"."ANODE CONVEYOR COVER FORWARD", signal13 := "PM07"."ANODE CONVEYOR COVER BACKWARD", signal14 := "PM07"."CATHODE CONVEYOR COVER FORWARD", signal15 := "PM07"."CATHODE CONVEYOR COVER BACKWARD", interfaceSignals := #statInterfaceSignalsHmi[56].valueSymbolLeft)
      #instSignals56Right(signal00 :=, signal01 :=, signal02 :=, signal03 :=, signal04 :=, signal05 :=, signal06 :=, signal07 :=, signal08 :=, signal09 :=, signal10 :=, signal11 :=, signal12 :=, signal13 :=, signal14 :=, signal15 :=, interfaceSignals := #statInterfaceSignalsHmi[56].valueSymbolRight)
   END_RUNG
   // the same network as SCL:
   #instSignals56Left(signal00 := "PM07"."JR WINDER CLAMP TOP REAR  UP",   // "LAF_InterfaceSignalsBool"
                      signal01 := "PM07"."JR WINDER CLAMP TOP REAR  DOWN",
                      signal02 := "PM07"."JR WINDER CLAMP BTM REAR UP",
                      signal03 := "PM07"."JR WINDER CLAMP BTM REAR DOWN",
                      signal04 := "PM07"."JR WINDER CLAMP TOP FRONT UP",
                      signal05 := "PM07"."JR WINDER CLAMP TOP FRONT DOWN",
                      signal06 := "PM07"."JR WINDER CLAMP BTM FRONT UP",
                      signal07 := "PM07"."JR WINDER CLAMP BTM FRONT DOWN",
                      signal08 := "PM07".SPARE,
                      signal09 := "PM07".SPARE_1,
                      signal10 := "PM07"."PUSH ROLLER FORWARD",
                      signal11 := "PM07"."PUSH ROLLER BACKWARD",
                      signal12 := "PM07"."ANODE CONVEYOR COVER FORWARD",
                      signal13 := "PM07"."ANODE CONVEYOR COVER BACKWARD",
                      signal14 := "PM07"."CATHODE CONVEYOR COVER FORWARD",
                      signal15 := "PM07"."CATHODE CONVEYOR COVER BACKWARD",
                      interfaceSignals := #statInterfaceSignalsHmi[56].valueSymbolLeft,
                      ENO => #_w1);
   IF #_w1 THEN
       #instSignals56Right(interfaceSignals := #statInterfaceSignalsHmi[56].valueSymbolRight);   // "LAF_InterfaceSignalsBool"
   END_IF;
END_REGION

REGION Network 62: Interface Signals 05 -Example: Model Flex-Pro-Line - IN/OUT- / Interface Signals 57
   // Aufruf des Schnittstellen Signal Bausteins Ba-Bereich 4 / Call the interface signals bool blocks of opmode 4
   RUNG wire#powerrail
      #instSignals57Left(signal00 := "SP201"."MAIN OP AUTO INITIATE PBL (GREEN)", signal01 := "SP201"."MAIN OP STOP PBL (RED)", signal02 := "SP201"."MAIN HMI POWER TRIPPED E110CB", signal03 :=, signal04 :=, signal05 :=, signal06 :=, signal07 :=, signal08 :=, signal09 :=, signal10 :=, signal11 :=, signal12 :=, signal13 :=, signal14 :=, signal15 :=, interfaceSignals := #statInterfaceSignalsHmi[57].valueSymbolLeft)
      #instSignals57Right(signal00 :=, signal01 :=, signal02 :=, signal03 :=, signal04 :=, signal05 :=, signal06 :=, signal07 :=, signal08 :=, signal09 :=, signal10 :=, signal11 :=, signal12 :=, signal13 :=, signal14 :=, signal15 :=, interfaceSignals := #statInterfaceSignalsHmi[57].valueSymbolRight)
   END_RUNG
   // the same network as SCL:
   #instSignals57Left(signal00 := "SP201"."MAIN OP AUTO INITIATE PBL (GREEN)",   // "LAF_InterfaceSignalsBool"
                      signal01 := "SP201"."MAIN OP STOP PBL (RED)",
                      signal02 := "SP201"."MAIN HMI POWER TRIPPED E110CB",
                      interfaceSignals := #statInterfaceSignalsHmi[57].valueSymbolLeft,
                      ENO => #_w1);
   IF #_w1 THEN
       #instSignals57Right(interfaceSignals := #statInterfaceSignalsHmi[57].valueSymbolRight);   // "LAF_InterfaceSignalsBool"
   END_IF;
END_REGION

REGION Network 63: Interface Signals 05 -Example: Model Flex-Pro-Line - IN/OUT- / Interface Signals 58
   // Aufruf des Schnittstellen Signal Bausteins Ba-Bereich 4 / Call the interface signals bool blocks of opmode 4
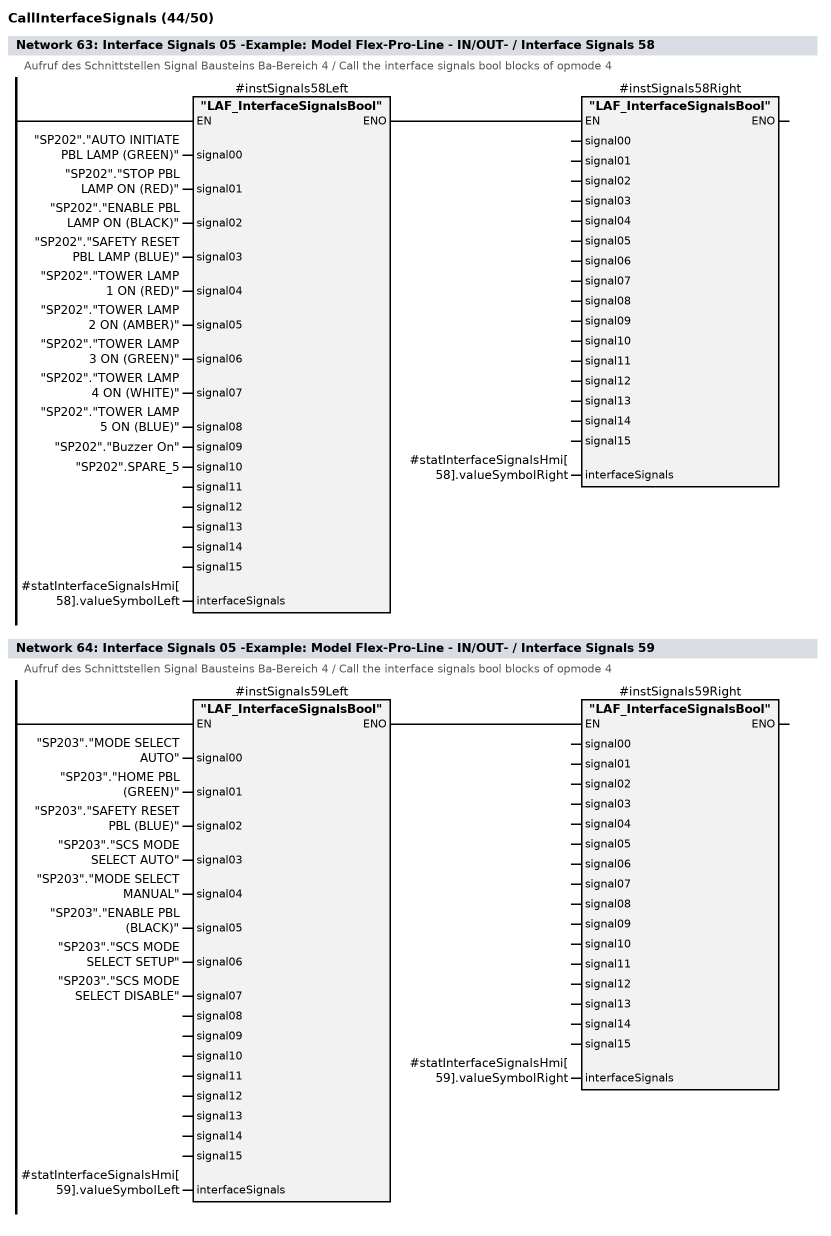
   RUNG wire#powerrail
      #instSignals58Left(signal00 := "SP202"."AUTO INITIATE PBL LAMP (GREEN)", signal01 := "SP202"."STOP PBL LAMP ON (RED)", signal02 := "SP202"."ENABLE PBL LAMP ON (BLACK)", signal03 := "SP202"."SAFETY RESET PBL LAMP (BLUE)", signal04 := "SP202"."TOWER LAMP 1 ON (RED)", signal05 := "SP202"."TOWER LAMP 2 ON (AMBER)", signal06 := "SP202"."TOWER LAMP 3 ON (GREEN)", signal07 := "SP202"."TOWER LAMP 4 ON (WHITE)", signal08 := "SP202"."TOWER LAMP 5 ON (BLUE)", signal09 := "SP202"."Buzzer On", signal10 := "SP202".SPARE_5, signal11 :=, signal12 :=, signal13 :=, signal14 :=, signal15 :=, interfaceSignals := #statInterfaceSignalsHmi[58].valueSymbolLeft)
      #instSignals58Right(signal00 :=, signal01 :=, signal02 :=, signal03 :=, signal04 :=, signal05 :=, signal06 :=, signal07 :=, signal08 :=, signal09 :=, signal10 :=, signal11 :=, signal12 :=, signal13 :=, signal14 :=, signal15 :=, interfaceSignals := #statInterfaceSignalsHmi[58].valueSymbolRight)
   END_RUNG
   // the same network as SCL:
   #instSignals58Left(signal00 := "SP202"."AUTO INITIATE PBL LAMP (GREEN)",   // "LAF_InterfaceSignalsBool"
                      signal01 := "SP202"."STOP PBL LAMP ON (RED)",
                      signal02 := "SP202"."ENABLE PBL LAMP ON (BLACK)",
                      signal03 := "SP202"."SAFETY RESET PBL LAMP (BLUE)",
                      signal04 := "SP202"."TOWER LAMP 1 ON (RED)",
                      signal05 := "SP202"."TOWER LAMP 2 ON (AMBER)",
                      signal06 := "SP202"."TOWER LAMP 3 ON (GREEN)",
                      signal07 := "SP202"."TOWER LAMP 4 ON (WHITE)",
                      signal08 := "SP202"."TOWER LAMP 5 ON (BLUE)",
                      signal09 := "SP202"."Buzzer On",
                      signal10 := "SP202".SPARE_5,
                      interfaceSignals := #statInterfaceSignalsHmi[58].valueSymbolLeft,
                      ENO => #_w1);
   IF #_w1 THEN
       #instSignals58Right(interfaceSignals := #statInterfaceSignalsHmi[58].valueSymbolRight);   // "LAF_InterfaceSignalsBool"
   END_IF;
END_REGION

REGION Network 64: Interface Signals 05 -Example: Model Flex-Pro-Line - IN/OUT- / Interface Signals 59
   // Aufruf des Schnittstellen Signal Bausteins Ba-Bereich 4 / Call the interface signals bool blocks of opmode 4
   RUNG wire#powerrail
      #instSignals59Left(signal00 := "SP203"."MODE SELECT AUTO", signal01 := "SP203"."HOME PBL (GREEN)", signal02 := "SP203"."SAFETY RESET PBL (BLUE)", signal03 := "SP203"."SCS MODE SELECT AUTO", signal04 := "SP203"."MODE SELECT MANUAL", signal05 := "SP203"."ENABLE PBL (BLACK)", signal06 := "SP203"."SCS MODE SELECT SETUP", signal07 := "SP203"."SCS MODE SELECT DISABLE", signal08 :=, signal09 :=, signal10 :=, signal11 :=, signal12 :=, signal13 :=, signal14 :=, signal15 :=, interfaceSignals := #statInterfaceSignalsHmi[59].valueSymbolLeft)
      #instSignals59Right(signal00 :=, signal01 :=, signal02 :=, signal03 :=, signal04 :=, signal05 :=, signal06 :=, signal07 :=, signal08 :=, signal09 :=, signal10 :=, signal11 :=, signal12 :=, signal13 :=, signal14 :=, signal15 :=, interfaceSignals := #statInterfaceSignalsHmi[59].valueSymbolRight)
   END_RUNG
   // the same network as SCL:
   #instSignals59Left(signal00 := "SP203"."MODE SELECT AUTO",   // "LAF_InterfaceSignalsBool"
                      signal01 := "SP203"."HOME PBL (GREEN)",
                      signal02 := "SP203"."SAFETY RESET PBL (BLUE)",
                      signal03 := "SP203"."SCS MODE SELECT AUTO",
                      signal04 := "SP203"."MODE SELECT MANUAL",
                      signal05 := "SP203"."ENABLE PBL (BLACK)",
                      signal06 := "SP203"."SCS MODE SELECT SETUP",
                      signal07 := "SP203"."SCS MODE SELECT DISABLE",
                      interfaceSignals := #statInterfaceSignalsHmi[59].valueSymbolLeft,
                      ENO => #_w1);
   IF #_w1 THEN
       #instSignals59Right(interfaceSignals := #statInterfaceSignalsHmi[59].valueSymbolRight);   // "LAF_InterfaceSignalsBool"
   END_IF;
END_REGION

REGION Network 65: Interface Signals 05 -Example: Model Flex-Pro-Line - IN/OUT- / Interface Signals 60
   // Aufruf des Schnittstellen Signal Bausteins Ba-Bereich 4 / Call the interface signals bool blocks of opmode 4
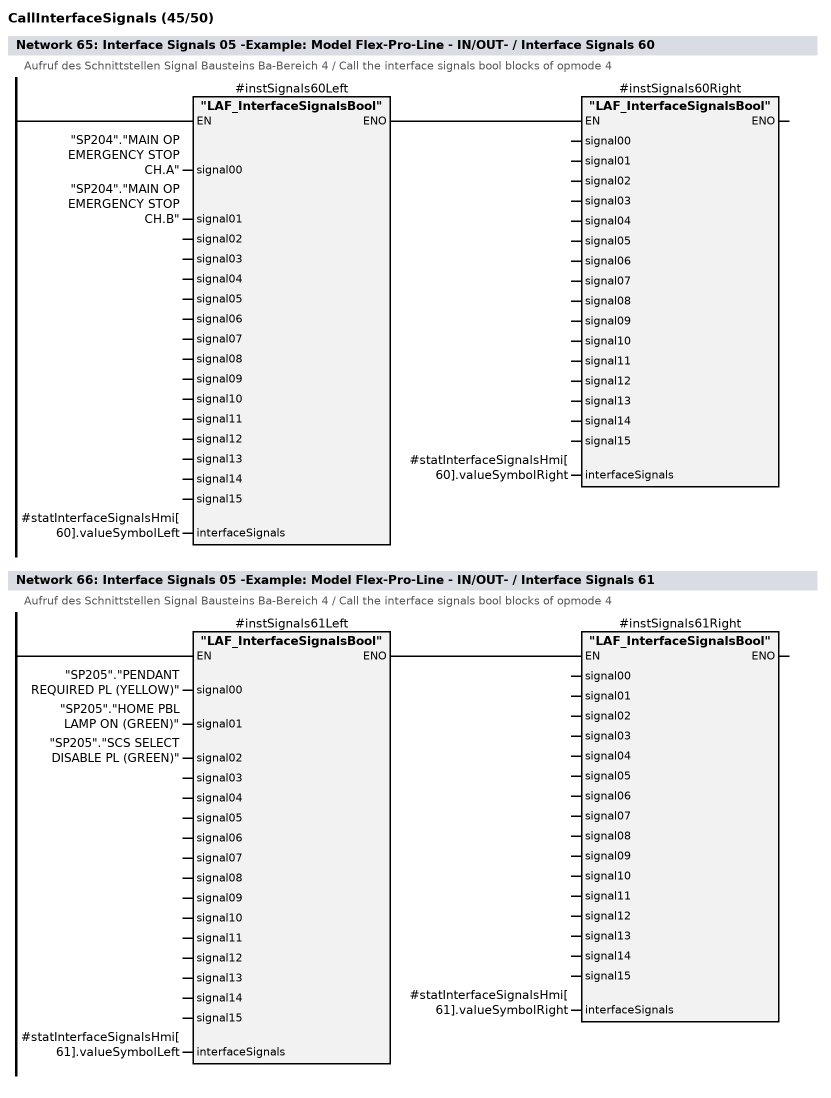
   RUNG wire#powerrail
      #instSignals60Left(signal00 := "SP204"."MAIN OP EMERGENCY STOP CH.A", signal01 := "SP204"."MAIN OP EMERGENCY STOP CH.B", signal02 :=, signal03 :=, signal04 :=, signal05 :=, signal06 :=, signal07 :=, signal08 :=, signal09 :=, signal10 :=, signal11 :=, signal12 :=, signal13 :=, signal14 :=, signal15 :=, interfaceSignals := #statInterfaceSignalsHmi[60].valueSymbolLeft)
      #instSignals60Right(signal00 :=, signal01 :=, signal02 :=, signal03 :=, signal04 :=, signal05 :=, signal06 :=, signal07 :=, signal08 :=, signal09 :=, signal10 :=, signal11 :=, signal12 :=, signal13 :=, signal14 :=, signal15 :=, interfaceSignals := #statInterfaceSignalsHmi[60].valueSymbolRight)
   END_RUNG
   // the same network as SCL:
   #instSignals60Left(signal00 := "SP204"."MAIN OP EMERGENCY STOP CH.A",   // "LAF_InterfaceSignalsBool"
                      signal01 := "SP204"."MAIN OP EMERGENCY STOP CH.B",
                      interfaceSignals := #statInterfaceSignalsHmi[60].valueSymbolLeft,
                      ENO => #_w1);
   IF #_w1 THEN
       #instSignals60Right(interfaceSignals := #statInterfaceSignalsHmi[60].valueSymbolRight);   // "LAF_InterfaceSignalsBool"
   END_IF;
END_REGION

REGION Network 66: Interface Signals 05 -Example: Model Flex-Pro-Line - IN/OUT- / Interface Signals 61
   // Aufruf des Schnittstellen Signal Bausteins Ba-Bereich 4 / Call the interface signals bool blocks of opmode 4
   RUNG wire#powerrail
      #instSignals61Left(signal00 := "SP205"."PENDANT REQUIRED PL (YELLOW)", signal01 := "SP205"."HOME PBL LAMP ON (GREEN)", signal02 := "SP205"."SCS SELECT DISABLE PL (GREEN)", signal03 :=, signal04 :=, signal05 :=, signal06 :=, signal07 :=, signal08 :=, signal09 :=, signal10 :=, signal11 :=, signal12 :=, signal13 :=, signal14 :=, signal15 :=, interfaceSignals := #statInterfaceSignalsHmi[61].valueSymbolLeft)
      #instSignals61Right(signal00 :=, signal01 :=, signal02 :=, signal03 :=, signal04 :=, signal05 :=, signal06 :=, signal07 :=, signal08 :=, signal09 :=, signal10 :=, signal11 :=, signal12 :=, signal13 :=, signal14 :=, signal15 :=, interfaceSignals := #statInterfaceSignalsHmi[61].valueSymbolRight)
   END_RUNG
   // the same network as SCL:
   #instSignals61Left(signal00 := "SP205"."PENDANT REQUIRED PL (YELLOW)",   // "LAF_InterfaceSignalsBool"
                      signal01 := "SP205"."HOME PBL LAMP ON (GREEN)",
                      signal02 := "SP205"."SCS SELECT DISABLE PL (GREEN)",
                      interfaceSignals := #statInterfaceSignalsHmi[61].valueSymbolLeft,
                      ENO => #_w1);
   IF #_w1 THEN
       #instSignals61Right(interfaceSignals := #statInterfaceSignalsHmi[61].valueSymbolRight);   // "LAF_InterfaceSignalsBool"
   END_IF;
END_REGION

REGION Network 67: Interface Signals 05 -Example: Model Flex-Pro-Line - IN/OUT- / Interface Signals 62
   // Aufruf des Schnittstellen Signal Bausteins Ba-Bereich 4 / Call the interface signals bool blocks of opmode 4
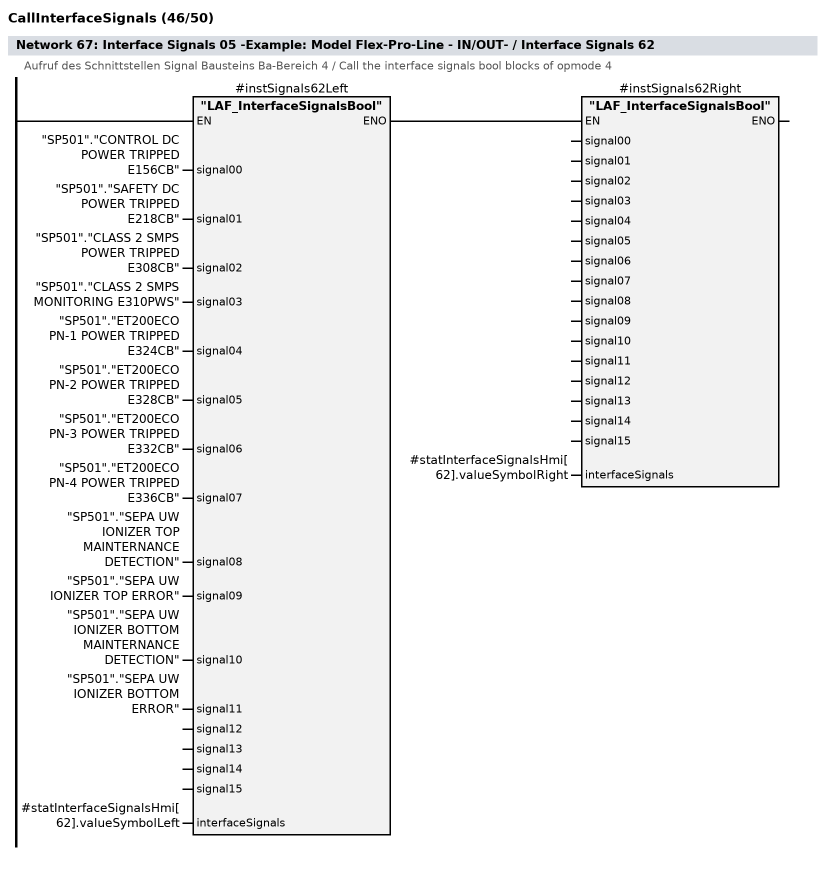
   RUNG wire#powerrail
      #instSignals62Left(signal00 := "SP501"."CONTROL DC POWER TRIPPED E156CB", signal01 := "SP501"."SAFETY DC POWER TRIPPED E218CB", signal02 := "SP501"."CLASS 2 SMPS POWER TRIPPED E308CB", signal03 := "SP501"."CLASS 2 SMPS MONITORING E310PWS", signal04 := "SP501"."ET200ECO PN-1 POWER TRIPPED E324CB", signal05 := "SP501"."ET200ECO PN-2 POWER TRIPPED E328CB", signal06 := "SP501"."ET200ECO PN-3 POWER TRIPPED E332CB", signal07 := "SP501"."ET200ECO PN-4 POWER TRIPPED E336CB", signal08 := "SP501"."SEPA UW IONIZER TOP MAINTERNANCE DETECTION", signal09 := "SP501"."SEPA UW IONIZER TOP ERROR", signal10 := "SP501"."SEPA UW IONIZER BOTTOM MAINTERNANCE DETECTION", signal11 := "SP501"."SEPA UW IONIZER BOTTOM ERROR", signal12 :=, signal13 :=, signal14 :=, signal15 :=, interfaceSignals := #statInterfaceSignalsHmi[62].valueSymbolLeft)
      #instSignals62Right(signal00 :=, signal01 :=, signal02 :=, signal03 :=, signal04 :=, signal05 :=, signal06 :=, signal07 :=, signal08 :=, signal09 :=, signal10 :=, signal11 :=, signal12 :=, signal13 :=, signal14 :=, signal15 :=, interfaceSignals := #statInterfaceSignalsHmi[62].valueSymbolRight)
   END_RUNG
   // the same network as SCL:
   #instSignals62Left(signal00 := "SP501"."CONTROL DC POWER TRIPPED E156CB",   // "LAF_InterfaceSignalsBool"
                      signal01 := "SP501"."SAFETY DC POWER TRIPPED E218CB",
                      signal02 := "SP501"."CLASS 2 SMPS POWER TRIPPED E308CB",
                      signal03 := "SP501"."CLASS 2 SMPS MONITORING E310PWS",
                      signal04 := "SP501"."ET200ECO PN-1 POWER TRIPPED E324CB",
                      signal05 := "SP501"."ET200ECO PN-2 POWER TRIPPED E328CB",
                      signal06 := "SP501"."ET200ECO PN-3 POWER TRIPPED E332CB",
                      signal07 := "SP501"."ET200ECO PN-4 POWER TRIPPED E336CB",
                      signal08 := "SP501"."SEPA UW IONIZER TOP MAINTERNANCE DETECTION",
                      signal09 := "SP501"."SEPA UW IONIZER TOP ERROR",
                      signal10 := "SP501"."SEPA UW IONIZER BOTTOM MAINTERNANCE DETECTION",
                      signal11 := "SP501"."SEPA UW IONIZER BOTTOM ERROR",
                      interfaceSignals := #statInterfaceSignalsHmi[62].valueSymbolLeft,
                      ENO => #_w1);
   IF #_w1 THEN
       #instSignals62Right(interfaceSignals := #statInterfaceSignalsHmi[62].valueSymbolRight);   // "LAF_InterfaceSignalsBool"
   END_IF;
END_REGION

REGION Network 68: Interface Signals 03 -Example: System flags & Clock flags- / Interface Signals63
   // Aufruf des Schnittstellen Signal Bausteins für die Systemvariablen / Call the interface signals bool blocks of system tags
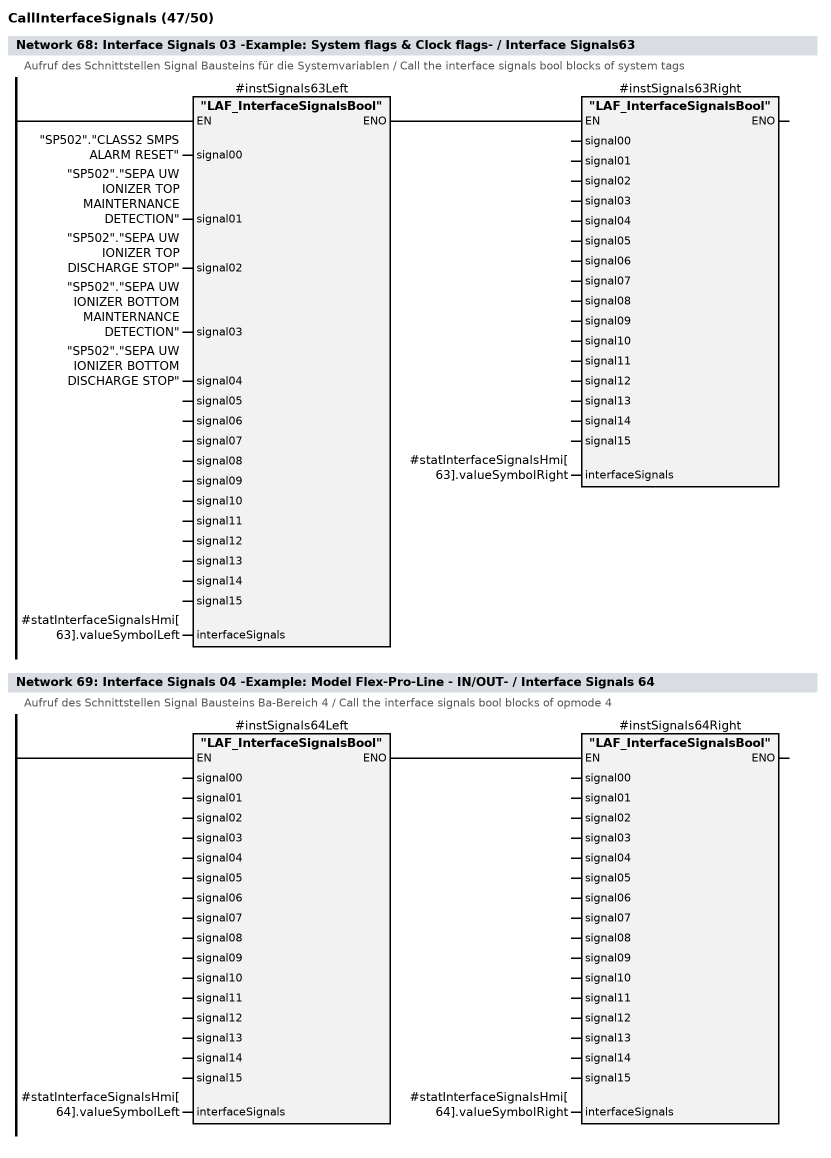
   RUNG wire#powerrail
      #instSignals63Left(signal00 := "SP502"."CLASS2 SMPS ALARM RESET", signal01 := "SP502"."SEPA UW IONIZER TOP MAINTERNANCE DETECTION", signal02 := "SP502"."SEPA UW IONIZER TOP DISCHARGE STOP", signal03 := "SP502"."SEPA UW IONIZER BOTTOM MAINTERNANCE DETECTION", signal04 := "SP502"."SEPA UW IONIZER BOTTOM DISCHARGE STOP", signal05 :=, signal06 :=, signal07 :=, signal08 :=, signal09 :=, signal10 :=, signal11 :=, signal12 :=, signal13 :=, signal14 :=, signal15 :=, interfaceSignals := #statInterfaceSignalsHmi[63].valueSymbolLeft)
      #instSignals63Right(signal00 :=, signal01 :=, signal02 :=, signal03 :=, signal04 :=, signal05 :=, signal06 :=, signal07 :=, signal08 :=, signal09 :=, signal10 :=, signal11 :=, signal12 :=, signal13 :=, signal14 :=, signal15 :=, interfaceSignals := #statInterfaceSignalsHmi[63].valueSymbolRight)
   END_RUNG
   // the same network as SCL:
   #instSignals63Left(signal00 := "SP502"."CLASS2 SMPS ALARM RESET",   // "LAF_InterfaceSignalsBool"
                      signal01 := "SP502"."SEPA UW IONIZER TOP MAINTERNANCE DETECTION",
                      signal02 := "SP502"."SEPA UW IONIZER TOP DISCHARGE STOP",
                      signal03 := "SP502"."SEPA UW IONIZER BOTTOM MAINTERNANCE DETECTION",
                      signal04 := "SP502"."SEPA UW IONIZER BOTTOM DISCHARGE STOP",
                      interfaceSignals := #statInterfaceSignalsHmi[63].valueSymbolLeft,
                      ENO => #_w1);
   IF #_w1 THEN
       #instSignals63Right(interfaceSignals := #statInterfaceSignalsHmi[63].valueSymbolRight);   // "LAF_InterfaceSignalsBool"
   END_IF;
END_REGION

REGION Network 69: Interface Signals 04 -Example: Model Flex-Pro-Line - IN/OUT- / Interface Signals 64
   // Aufruf des Schnittstellen Signal Bausteins Ba-Bereich 4 / Call the interface signals bool blocks of opmode 4
   RUNG wire#powerrail
      #instSignals64Left(signal00 :=, signal01 :=, signal02 :=, signal03 :=, signal04 :=, signal05 :=, signal06 :=, signal07 :=, signal08 :=, signal09 :=, signal10 :=, signal11 :=, signal12 :=, signal13 :=, signal14 :=, signal15 :=, interfaceSignals := #statInterfaceSignalsHmi[64].valueSymbolLeft)
      #instSignals64Right(signal00 :=, signal01 :=, signal02 :=, signal03 :=, signal04 :=, signal05 :=, signal06 :=, signal07 :=, signal08 :=, signal09 :=, signal10 :=, signal11 :=, signal12 :=, signal13 :=, signal14 :=, signal15 :=, interfaceSignals := #statInterfaceSignalsHmi[64].valueSymbolRight)
   END_RUNG
   // the same network as SCL:
   #instSignals64Left(interfaceSignals := #statInterfaceSignalsHmi[64].valueSymbolLeft, ENO => #_w1);   // "LAF_InterfaceSignalsBool"
   IF #_w1 THEN
       #instSignals64Right(interfaceSignals := #statInterfaceSignalsHmi[64].valueSymbolRight);   // "LAF_InterfaceSignalsBool"
   END_IF;
END_REGION

REGION Network 70: Interface Signals 05 -Example: Model Flex-Pro-Line - IN/OUT- / Interface Signals 65
   // Aufruf des Schnittstellen Signal Bausteins Ba-Bereich 4 / Call the interface signals bool blocks of opmode 4
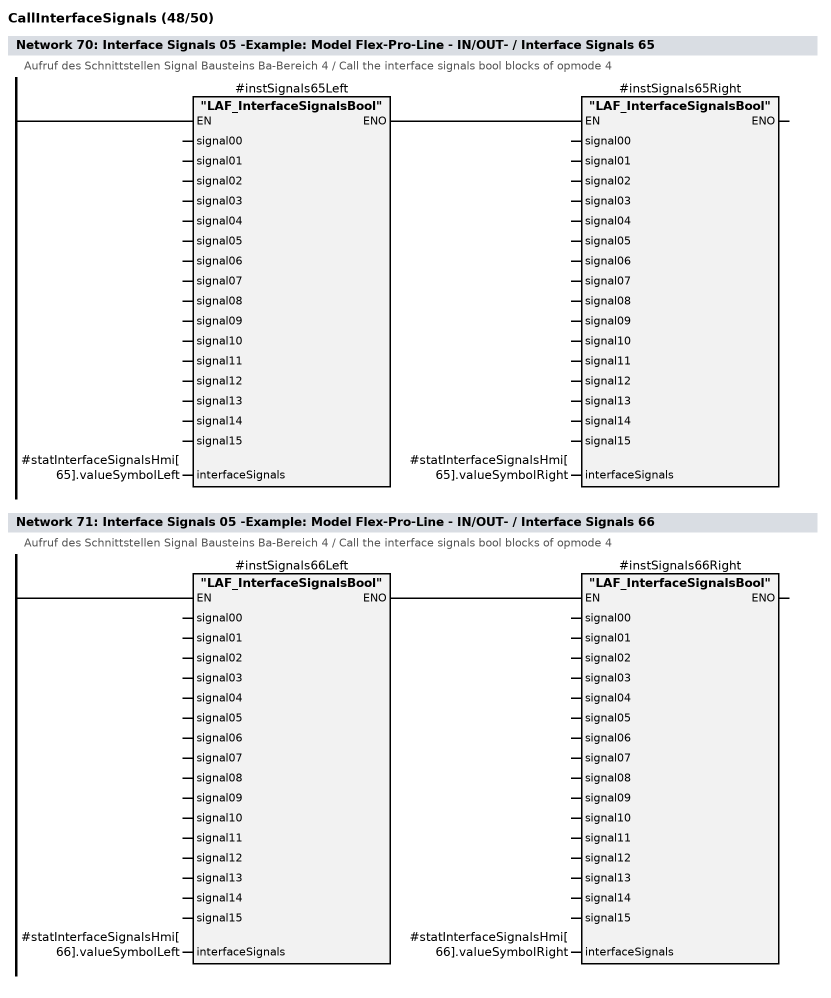
   RUNG wire#powerrail
      #instSignals65Left(signal00 :=, signal01 :=, signal02 :=, signal03 :=, signal04 :=, signal05 :=, signal06 :=, signal07 :=, signal08 :=, signal09 :=, signal10 :=, signal11 :=, signal12 :=, signal13 :=, signal14 :=, signal15 :=, interfaceSignals := #statInterfaceSignalsHmi[65].valueSymbolLeft)
      #instSignals65Right(signal00 :=, signal01 :=, signal02 :=, signal03 :=, signal04 :=, signal05 :=, signal06 :=, signal07 :=, signal08 :=, signal09 :=, signal10 :=, signal11 :=, signal12 :=, signal13 :=, signal14 :=, signal15 :=, interfaceSignals := #statInterfaceSignalsHmi[65].valueSymbolRight)
   END_RUNG
   // the same network as SCL:
   #instSignals65Left(interfaceSignals := #statInterfaceSignalsHmi[65].valueSymbolLeft, ENO => #_w1);   // "LAF_InterfaceSignalsBool"
   IF #_w1 THEN
       #instSignals65Right(interfaceSignals := #statInterfaceSignalsHmi[65].valueSymbolRight);   // "LAF_InterfaceSignalsBool"
   END_IF;
END_REGION

REGION Network 71: Interface Signals 05 -Example: Model Flex-Pro-Line - IN/OUT- / Interface Signals 66
   // Aufruf des Schnittstellen Signal Bausteins Ba-Bereich 4 / Call the interface signals bool blocks of opmode 4
   RUNG wire#powerrail
      #instSignals66Left(signal00 :=, signal01 :=, signal02 :=, signal03 :=, signal04 :=, signal05 :=, signal06 :=, signal07 :=, signal08 :=, signal09 :=, signal10 :=, signal11 :=, signal12 :=, signal13 :=, signal14 :=, signal15 :=, interfaceSignals := #statInterfaceSignalsHmi[66].valueSymbolLeft)
      #instSignals66Right(signal00 :=, signal01 :=, signal02 :=, signal03 :=, signal04 :=, signal05 :=, signal06 :=, signal07 :=, signal08 :=, signal09 :=, signal10 :=, signal11 :=, signal12 :=, signal13 :=, signal14 :=, signal15 :=, interfaceSignals := #statInterfaceSignalsHmi[66].valueSymbolRight)
   END_RUNG
   // the same network as SCL:
   #instSignals66Left(interfaceSignals := #statInterfaceSignalsHmi[66].valueSymbolLeft, ENO => #_w1);   // "LAF_InterfaceSignalsBool"
   IF #_w1 THEN
       #instSignals66Right(interfaceSignals := #statInterfaceSignalsHmi[66].valueSymbolRight);   // "LAF_InterfaceSignalsBool"
   END_IF;
END_REGION

REGION Network 72: Interface Signals 05 -Example: Model Flex-Pro-Line - IN/OUT- / Interface Signals 67
   // Aufruf des Schnittstellen Signal Bausteins Ba-Bereich 4 / Call the interface signals bool blocks of opmode 4
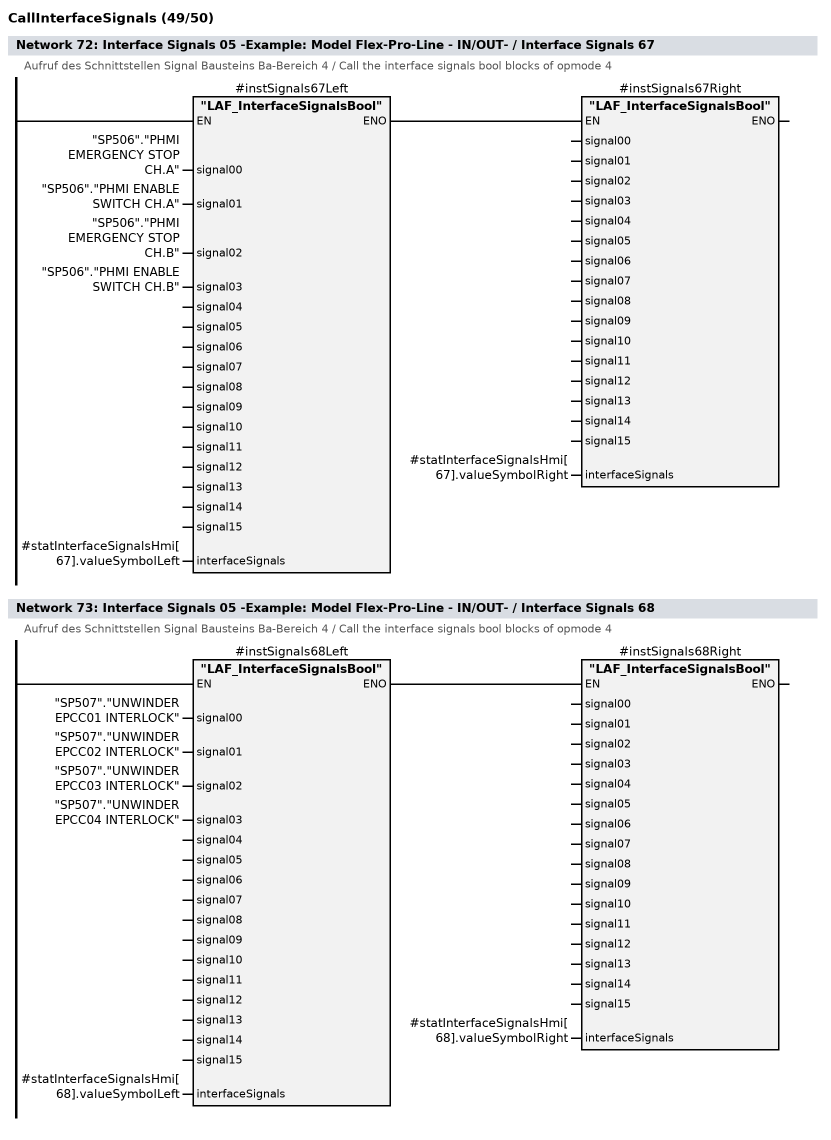
   RUNG wire#powerrail
      #instSignals67Left(signal00 := "SP506"."PHMI EMERGENCY STOP CH.A", signal01 := "SP506"."PHMI ENABLE SWITCH CH.A", signal02 := "SP506"."PHMI EMERGENCY STOP CH.B", signal03 := "SP506"."PHMI ENABLE SWITCH CH.B", signal04 :=, signal05 :=, signal06 :=, signal07 :=, signal08 :=, signal09 :=, signal10 :=, signal11 :=, signal12 :=, signal13 :=, signal14 :=, signal15 :=, interfaceSignals := #statInterfaceSignalsHmi[67].valueSymbolLeft)
      #instSignals67Right(signal00 :=, signal01 :=, signal02 :=, signal03 :=, signal04 :=, signal05 :=, signal06 :=, signal07 :=, signal08 :=, signal09 :=, signal10 :=, signal11 :=, signal12 :=, signal13 :=, signal14 :=, signal15 :=, interfaceSignals := #statInterfaceSignalsHmi[67].valueSymbolRight)
   END_RUNG
   // the same network as SCL:
   #instSignals67Left(signal00 := "SP506"."PHMI EMERGENCY STOP CH.A",   // "LAF_InterfaceSignalsBool"
                      signal01 := "SP506"."PHMI ENABLE SWITCH CH.A",
                      signal02 := "SP506"."PHMI EMERGENCY STOP CH.B",
                      signal03 := "SP506"."PHMI ENABLE SWITCH CH.B",
                      interfaceSignals := #statInterfaceSignalsHmi[67].valueSymbolLeft,
                      ENO => #_w1);
   IF #_w1 THEN
       #instSignals67Right(interfaceSignals := #statInterfaceSignalsHmi[67].valueSymbolRight);   // "LAF_InterfaceSignalsBool"
   END_IF;
END_REGION

REGION Network 73: Interface Signals 05 -Example: Model Flex-Pro-Line - IN/OUT- / Interface Signals 68
   // Aufruf des Schnittstellen Signal Bausteins Ba-Bereich 4 / Call the interface signals bool blocks of opmode 4
   RUNG wire#powerrail
      #instSignals68Left(signal00 := "SP507"."UNWINDER EPCC01 INTERLOCK", signal01 := "SP507"."UNWINDER EPCC02 INTERLOCK", signal02 := "SP507"."UNWINDER EPCC03 INTERLOCK", signal03 := "SP507"."UNWINDER EPCC04 INTERLOCK", signal04 :=, signal05 :=, signal06 :=, signal07 :=, signal08 :=, signal09 :=, signal10 :=, signal11 :=, signal12 :=, signal13 :=, signal14 :=, signal15 :=, interfaceSignals := #statInterfaceSignalsHmi[68].valueSymbolLeft)
      #instSignals68Right(signal00 :=, signal01 :=, signal02 :=, signal03 :=, signal04 :=, signal05 :=, signal06 :=, signal07 :=, signal08 :=, signal09 :=, signal10 :=, signal11 :=, signal12 :=, signal13 :=, signal14 :=, signal15 :=, interfaceSignals := #statInterfaceSignalsHmi[68].valueSymbolRight)
   END_RUNG
   // the same network as SCL:
   #instSignals68Left(signal00 := "SP507"."UNWINDER EPCC01 INTERLOCK",   // "LAF_InterfaceSignalsBool"
                      signal01 := "SP507"."UNWINDER EPCC02 INTERLOCK",
                      signal02 := "SP507"."UNWINDER EPCC03 INTERLOCK",
                      signal03 := "SP507"."UNWINDER EPCC04 INTERLOCK",
                      interfaceSignals := #statInterfaceSignalsHmi[68].valueSymbolLeft,
                      ENO => #_w1);
   IF #_w1 THEN
       #instSignals68Right(interfaceSignals := #statInterfaceSignalsHmi[68].valueSymbolRight);   // "LAF_InterfaceSignalsBool"
   END_IF;
END_REGION

REGION Network 74: Interface Signals 05 -Example: Model Flex-Pro-Line - IN/OUT- / Interface Signals 69
   // Aufruf des Schnittstellen Signal Bausteins Ba-Bereich 4 / Call the interface signals bool blocks of opmode 4
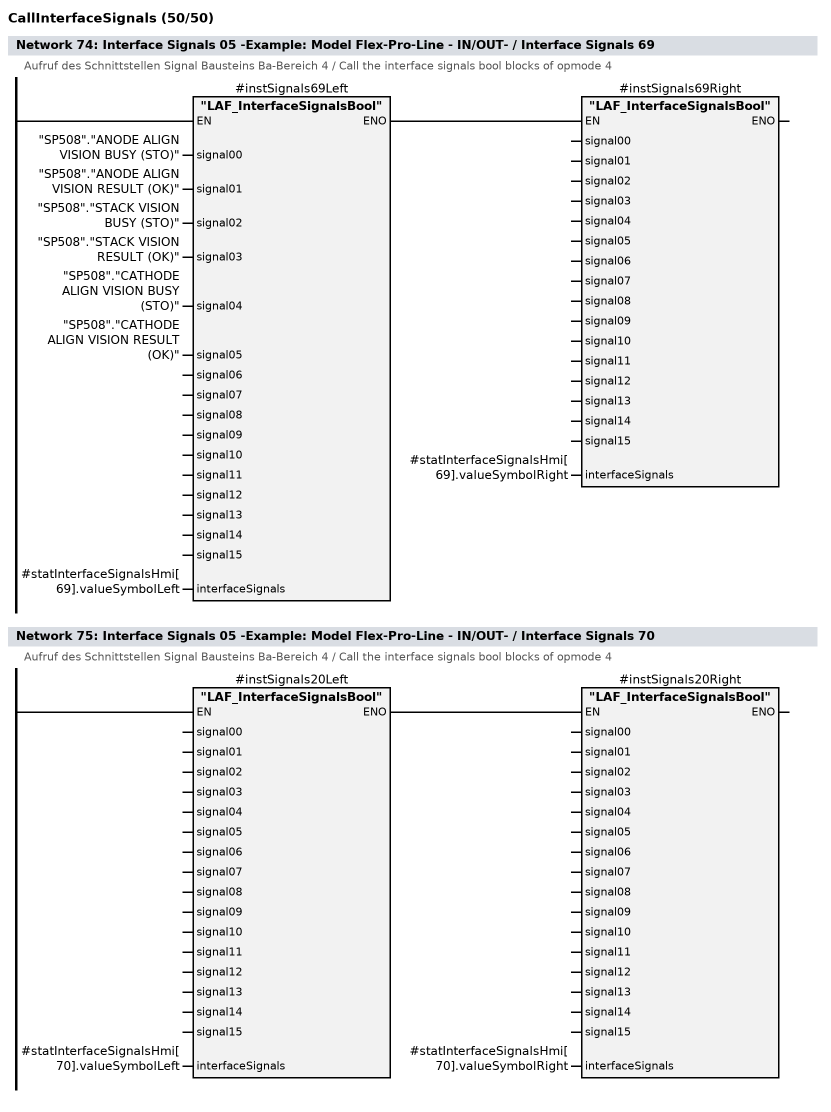
   RUNG wire#powerrail
      #instSignals69Left(signal00 := "SP508"."ANODE ALIGN VISION BUSY (STO)", signal01 := "SP508"."ANODE ALIGN VISION RESULT (OK)", signal02 := "SP508"."STACK VISION BUSY (STO)", signal03 := "SP508"."STACK VISION RESULT (OK)", signal04 := "SP508"."CATHODE ALIGN VISION BUSY (STO)", signal05 := "SP508"."CATHODE ALIGN VISION RESULT (OK)", signal06 :=, signal07 :=, signal08 :=, signal09 :=, signal10 :=, signal11 :=, signal12 :=, signal13 :=, signal14 :=, signal15 :=, interfaceSignals := #statInterfaceSignalsHmi[69].valueSymbolLeft)
      #instSignals69Right(signal00 :=, signal01 :=, signal02 :=, signal03 :=, signal04 :=, signal05 :=, signal06 :=, signal07 :=, signal08 :=, signal09 :=, signal10 :=, signal11 :=, signal12 :=, signal13 :=, signal14 :=, signal15 :=, interfaceSignals := #statInterfaceSignalsHmi[69].valueSymbolRight)
   END_RUNG
   // the same network as SCL:
   #instSignals69Left(signal00 := "SP508"."ANODE ALIGN VISION BUSY (STO)",   // "LAF_InterfaceSignalsBool"
                      signal01 := "SP508"."ANODE ALIGN VISION RESULT (OK)",
                      signal02 := "SP508"."STACK VISION BUSY (STO)",
                      signal03 := "SP508"."STACK VISION RESULT (OK)",
                      signal04 := "SP508"."CATHODE ALIGN VISION BUSY (STO)",
                      signal05 := "SP508"."CATHODE ALIGN VISION RESULT (OK)",
                      interfaceSignals := #statInterfaceSignalsHmi[69].valueSymbolLeft,
                      ENO => #_w1);
   IF #_w1 THEN
       #instSignals69Right(interfaceSignals := #statInterfaceSignalsHmi[69].valueSymbolRight);   // "LAF_InterfaceSignalsBool"
   END_IF;
END_REGION

REGION Network 75: Interface Signals 05 -Example: Model Flex-Pro-Line - IN/OUT- / Interface Signals 70
   // Aufruf des Schnittstellen Signal Bausteins Ba-Bereich 4 / Call the interface signals bool blocks of opmode 4
   RUNG wire#powerrail
      #instSignals20Left(signal00 :=, signal01 :=, signal02 :=, signal03 :=, signal04 :=, signal05 :=, signal06 :=, signal07 :=, signal08 :=, signal09 :=, signal10 :=, signal11 :=, signal12 :=, signal13 :=, signal14 :=, signal15 :=, interfaceSignals := #statInterfaceSignalsHmi[70].valueSymbolLeft)
      #instSignals20Right(signal00 :=, signal01 :=, signal02 :=, signal03 :=, signal04 :=, signal05 :=, signal06 :=, signal07 :=, signal08 :=, signal09 :=, signal10 :=, signal11 :=, signal12 :=, signal13 :=, signal14 :=, signal15 :=, interfaceSignals := #statInterfaceSignalsHmi[70].valueSymbolRight)
   END_RUNG
   // the same network as SCL:
   #instSignals20Left(interfaceSignals := #statInterfaceSignalsHmi[70].valueSymbolLeft, ENO => #_w1);   // "LAF_InterfaceSignalsBool"
   IF #_w1 THEN
       #instSignals20Right(interfaceSignals := #statInterfaceSignalsHmi[70].valueSymbolRight);   // "LAF_InterfaceSignalsBool"
   END_IF;
END_REGION
END_FUNCTION_BLOCK

FUNCTION_BLOCK "CallInterfaceSignalsConv"   // FB106, LAD
// stored: MemoryReserve 100, SetENOAutomatically false
   VAR_INPUT
      InterfaceTestMode : Bool;
   END_VAR
   VAR_OUTPUT
      signalsS2R : "typeReelCutToStack";
      signalsR2S : "typeStackToReelCut";
   END_VAR
   VAR_IN_OUT
      CommS2R : Array[0..95] of Bool;
      CommR2S : Array[0..95] of Bool;
      InterfaceTestButton : "LER_SignalsInput";
   END_VAR
   VAR
      statWordBuffer_2 { S7_SetPoint := 'True'} : Array[0..5] of Word;
      statWordBuffer_1 : Array[0..5] of Word;
   END_VAR
   VAR_TEMP
      tempDeleteData : "LER_SignalsInput";
   END_VAR
   VAR CONSTANT
      TRUE : Bool := TRUE;
   END_VAR
   VAR_TEMP   // added for the SCL form of the ladder/FBD networks
      _w1 : Bool;
      _w2 : Bool;
      _w3 : Bool;
      _w4 : Bool;
   END_VAR
BEGIN

REGION Network 1: CommR2S -> signalsR2S
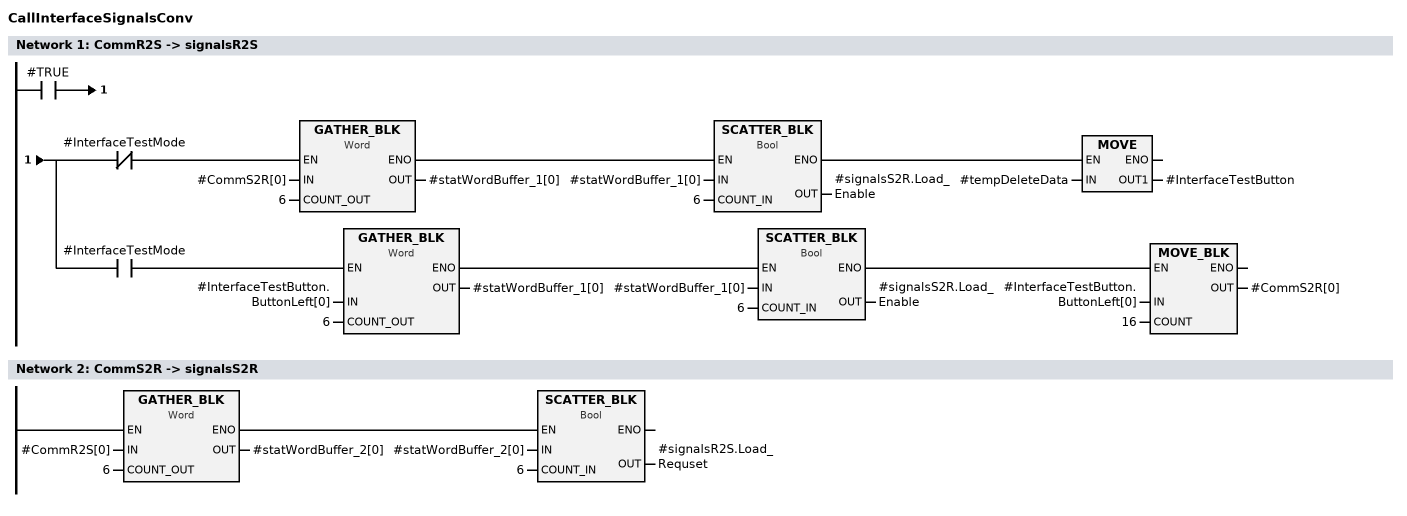
   GATHER_BLK(EN := #TRUE AND NOT #InterfaceTestMode,
              IN := #CommS2R[0],
              COUNT_OUT := 6,
              OUT => #statWordBuffer_1[0],
              ENO => #_w1);
   SCATTER_BLK(EN := #_w1,
               IN := #statWordBuffer_1[0],
               COUNT_IN := 6,
               OUT => #signalsS2R.Load_Enable,
               ENO => #_w2);
   IF #_w2 THEN #InterfaceTestButton := #tempDeleteData; END_IF;
   GATHER_BLK(EN := #TRUE AND #InterfaceTestMode,
              IN := #InterfaceTestButton.ButtonLeft[0],
              COUNT_OUT := 6,
              OUT => #statWordBuffer_1[0],
              ENO => #_w3);
   SCATTER_BLK(EN := #_w3,
               IN := #statWordBuffer_1[0],
               COUNT_IN := 6,
               OUT => #signalsS2R.Load_Enable,
               ENO => #_w4);
   IF #_w4 THEN MOVE_BLK(IN := #InterfaceTestButton.ButtonLeft[0], COUNT := 16, OUT => #CommS2R[0]); END_IF;
END_REGION

REGION Network 2: CommS2R -> signalsS2R
   RUNG wire#powerrail
      { S7_Templates := "[dest_type := Word, src_type := Bool, count_type := UInt]" } GATHER_BLK(IN := #CommR2S[0], COUNT_OUT := 6, OUT => #statWordBuffer_2[0])
      { S7_Templates := "[dest_type := Bool, src_type := Word, count_type := UInt]" } SCATTER_BLK(IN := #statWordBuffer_2[0], COUNT_IN := 6, OUT => #signalsR2S.Load_Requset)
   END_RUNG
   // the same network as SCL:
   GATHER_BLK(IN := #CommR2S[0], COUNT_OUT := 6, OUT => #statWordBuffer_2[0], ENO => #_w1);
   IF #_w1 THEN
       SCATTER_BLK(IN := #statWordBuffer_2[0], COUNT_IN := 6, OUT => #signalsR2S.Load_Requset);
   END_IF;
END_REGION
END_FUNCTION_BLOCK

FUNCTION_BLOCK "GetMotorstarterSignals"
{ S7_Optimized_Access := 'TRUE' ; Published := 'FALSE' }
VERSION : 0.1
   VAR_INPUT 
      Et200SpMotorstarterInterfaceAllUnits { ExternalAccessible := 'False'; ExternalVisible := 'False'; ExternalWritable := 'False'} : Array[0.."NO_OF_UNITS"] of "typeEmMotorStarterInterface";   // HMI: motorstarter values
      numberOfMS : USInt;
   END_VAR

   VAR_OUTPUT 
      selectedUnit : USInt;
      selectedEM : USInt;
      error : Word;
   END_VAR

   VAR_IN_OUT 
      Et200SpMotorstarterInterfaceHmi : "typeEt200SpMotorstarterInterfaceHmi";
   END_VAR

   VAR 
      statSelectedEMMotorStarter : USInt := 1;
      statSelectedUnitMotorStarter : USInt := 1;   // HMI: Selected unit
   END_VAR

   VAR_TEMP 
      tempEnable : Bool;   // Temporary value for input 'enable'
      tempEt200SpMotorstarterCurrent : Array[0.."NO_OF_ET200SPMOTORSTARTER"] of Real;
      tempEt200SpMotorstarterInputs : Array[0.."NO_OF_ET200SPMOTORSTARTER"] of "LSicar_typeMotorstarterIn";
      tempEt200SpMotorstarterOutputs : Array[0.."NO_OF_ET200SPMOTORSTARTER"] of "LSicar_typeMotorstarterOut";
      tempIndexMotorstarter : USInt;
      tempNoOfMS : USInt;
   END_VAR

   VAR CONSTANT 
      "INVALID UNIT" : Word := 16#7001;   // non existant unit
      "INVALID EM" : Word := 16#7002;   // non existant em
      OK : Word := 16#7000;
   END_VAR


BEGIN
	REGION BLOCK INFO HEADER
	    //===============================================================================
	    // Siemens AG / (c)Copyright 2024
	    //-------------------------------------------------------------------------------
	    // Title:            LAF_GetMotorstarterSignals
	    // Comment/Function: This block reads diagnostic information of a Motorstarter depending
	    //                   on the unit and Control Module selected in the HMI by the user.
	    // Library/Family:   Automation Framework / Motorstarter Diagnostic
	    // Author:           Siemens Digital Industries
	    // Tested with:      S7-1517TF V3.1
	    // Engineering:      TIA Portal V19
	    // Restrictions:     
	    //                   Required UDTs: LAF_typeDriveDiagConfig, LAF_typeDriveDiagInterfaceHmi
	    // Requirements:     S7-1500(T), MC_Version V8.0
	    //-------------------------------------------------------------------------------
	    // Change log table:
	    // Version  | Date       | Expert in charge        | Changes applied
	    //----------|------------|-------------------------|-----------------------------
	    // 01.00.00 | 05.06.2024 | SIMATIC Systems Support | First released version
	    //===============================================================================
	END_REGION BLOCK INFO HEADER
	
	REGION DESCRIPTION
	(/*
	This block reads diagnostic information (control inputs and outputs) of a Motorstarter. 
	At runtime, this block is enabled when the ET200SP Motorstarter screen is shown in the HMI. 
	Based on the selected motorstarter object in the HMI by the user. The shown information in the HMI depends on the
	Unit and Cotrol Module selected. 
	*/)
	END_REGION DESCRIPTION
	
	REGION INPUTS
	    //working with static values to keep the last selected value when opening for the first time the screen  
	  
	    #statSelectedUnitMotorStarter := #Et200SpMotorstarterInterfaceHmi.et200SpUnitMotorstarter;
	    #statSelectedEMMotorStarter := #Et200SpMotorstarterInterfaceHmi.et200SpEMMotorstarter;
	
	END_REGION INPUTS
	
	REGION ASSIGNING TEMPORARY VALUES
	    // Statement section REGION
	    IF #statSelectedUnitMotorStarter <= "NO_OF_UNITS" THEN
	        IF #statSelectedEMMotorStarter < "NO_OF_EM" THEN
	            #tempEt200SpMotorstarterCurrent := #Et200SpMotorstarterInterfaceAllUnits[#statSelectedUnitMotorStarter].EMmotorstarter[#statSelectedEMMotorStarter].et200SpMotorstarterCurrent;
	            #tempEt200SpMotorstarterInputs := #Et200SpMotorstarterInterfaceAllUnits[#statSelectedUnitMotorStarter].EMmotorstarter[#statSelectedEMMotorStarter].et200SpMotorstarterInputs;
	            #tempEt200SpMotorstarterOutputs := #Et200SpMotorstarterInterfaceAllUnits[#statSelectedUnitMotorStarter].EMmotorstarter[#statSelectedEMMotorStarter].et200SpMotorstarterOutputs;
	            #tempNoOfMS := #numberOfMS;
	            #error := #OK;
	        ELSE
	            #error := #"INVALID EM";
	        END_IF;
	
	    ELSE
	        #error := #"INVALID UNIT";
	    END_IF;
	
	
	END_REGION
	
	
	REGION OUTPUTS
	    // Statement section REGION
	    #Et200SpMotorstarterInterfaceHmi.et200SpMotorstarterCurrent := #tempEt200SpMotorstarterCurrent;
	    #Et200SpMotorstarterInterfaceHmi.et200SpMotorstarterInputs := #tempEt200SpMotorstarterInputs;
	    #Et200SpMotorstarterInterfaceHmi.et200SpMotorstarterOutputs := #tempEt200SpMotorstarterOutputs;
	    #Et200SpMotorstarterInterfaceHmi.et200SpNumberOfMotorstarters := #tempNoOfMS;
	    #selectedEM := #statSelectedEMMotorStarter;
	    #selectedUnit := #statSelectedUnitMotorStarter;
	END_REGION
	
	
END_FUNCTION_BLOCK

FUNCTION "DemoIdentRf" : Void   // FC79, LAD
TITLE = Demo: IDENT_FC / Demo: Ident
AUTHOR : SICAR
FAMILY : Demo
VERSION : 1.0
// Demo fuer Anwendung Ident Bausteine / Demo for usage of ident moduls
// stored: IsIECCheckEnabled true, SetENOAutomatically true
   // Ret_Val : Ret_Val
BEGIN

REGION Network 1: Änderungshistorie / ChangeLog
   // Die Änderungshistorie wird nur in englischer Editiersprache geführt.
   // Change log table:
   // Version | Date | Expert in charge | Changes applied
   // -------|---------|-------------|--------------------------------------------
   // 05.00.00 | 01.09.2023 | SICAR | First released version
END_REGION

REGION Network 2: Schreiben reader 1 / Define reading informations
   // Schreibe den String "Siemens" in die zu schreibende Datenstrucktur des RFID Geräts / Write the String "Siemens" in the writting structur of the FB
END_REGION

REGION Network 3: Schreiben reader 1 / Define writting informations
   // Schreibe den String "Siemens" in die zu schreibende Datenstrucktur des RFID Geräts / Write the String "Automation Framework" in the writting structur of the FB
END_REGION

REGION Network 4: Schreiben reader 1 / Define reading informations
   // Schreibe den String "Siemens" in die zu schreibende Datenstrucktur des RFID Geräts / Write the String "RF2385-621863" in the writting structur of the FB
END_REGION

REGION Network 5: Schreiben reader 1 / Define reading informations
   // Schreibe den String "Siemens" in die zu schreibende Datenstrucktur des RFID Geräts / Write the String "Demo RFID" in the writting structur of the FB
END_REGION
END_FUNCTION

FUNCTION_BLOCK "GetIdentRf"
{ S7_Optimized_Access := 'TRUE' ; Published := 'TRUE' }
VERSION : 0.1
   VAR_INPUT 
      identRfAllUnits { ExternalAccessible := 'False'; ExternalVisible := 'False'; ExternalWritable := 'False'} : Array[0.."NO_OF_UNITS"] of "typeEMIdentRf";   // HMI: motorstarter values
      numberOfRfReaders : USInt;
   END_VAR

   VAR_OUTPUT 
      selectedUnit : USInt := 1;
      selectedEM : USInt;
      error : Word;
   END_VAR

   VAR_IN_OUT 
      IdentRfInterfaceHmi : "typeIdentRfHmi";
   END_VAR

   VAR 
      statSelectedEMIdentRf : USInt := 1;
      statSelectedUnitIdentRf : USInt := 1;   // HMI: Selected unit
   END_VAR

   VAR_TEMP 
      tempEnable : Bool;   // Temporary value for input 'enable'
      tempRfReader : Array[0.."NO_OF_RF_IDENT_DEVICES"] of "LSicar_typeIdentInterfaceHmi";
      tempIndexIdentRf : USInt;
      tempNoOfidertRf : USInt;
   END_VAR

   VAR CONSTANT 
      "INVALID UNIT" : Word := 16#7001;   // non existant unit
      "INVALID EM" : Word := 16#7002;   // non existant em
      OK : Word := 16#7000;
   END_VAR


BEGIN
	REGION BLOCK INFO HEADER
	    //===============================================================================
	    // Siemens AG / (c)Copyright 2024
	    //-------------------------------------------------------------------------------
	    // Title:            LAF_GetMotorstarterSignals
	    // Comment/Function: This block reads diagnostic information of a Motorstarter depending
	    //                   on the unit and Control Module selected in the HMI by the user.
	    // Library/Family:   Automation Framework / Motorstarter Diagnostic
	    // Author:           Siemens Digital Industries
	    // Tested with:      S7-1517TF V3.1
	    // Engineering:      TIA Portal V19
	    // Restrictions:     
	    //                   Required UDTs: LAF_typeDriveDiagConfig, LAF_typeDriveDiagInterfaceHmi
	    // Requirements:     S7-1500(T), MC_Version V8.0
	    //-------------------------------------------------------------------------------
	    // Change log table:
	    // Version  | Date       | Expert in charge        | Changes applied
	    //----------|------------|-------------------------|-----------------------------
	    // 01.00.00 | 05.06.2024 | SIMATIC Systems Support | First released version
	    //===============================================================================
	END_REGION BLOCK INFO HEADER
	
	REGION DESCRIPTION
	(/*
	This block reads diagnostic information (control inputs and outputs) of a Motorstarter. 
	At runtime, this block is enabled when the ET200SP Motorstarter screen is shown in the HMI. 
	Based on the selected motorstarter object in the HMI by the user. The shown information in the HMI depends on the
	Unit and Cotrol Module selected. 
	*/)
	END_REGION DESCRIPTION
	
	REGION INPUTS
	    //working with static values to keep the last selected value when opening for the first time the screen  
	  
	    #statSelectedUnitIdentRf := #IdentRfInterfaceHmi.selectedUnit;
	    #statSelectedEMIdentRf := #IdentRfInterfaceHmi.selectedEM;
	
	END_REGION INPUTS
	
	REGION ASSIGNING TEMPORARY VALUES
	    // Statement section REGION
	    IF #statSelectedUnitIdentRf <= "NO_OF_UNITS" THEN
	        IF #statSelectedEMIdentRf < "NO_OF_EM" THEN
	            #tempRfReader:= #identRfAllUnits[#statSelectedUnitIdentRf].identRfEM[#statSelectedEMIdentRf].rfReader;
	            #tempNoOfidertRf := #numberOfRfReaders;
	             #error := #OK;
	        ELSE
	            #error := #"INVALID EM";
	        END_IF;
	
	    ELSE
	        #error := #"INVALID UNIT";
	    END_IF;
	
	
	END_REGION
	
	
	REGION OUTPUTS
	    // Statement section REGION
	    #IdentRfInterfaceHmi.rfReader := #tempRfReader;
	    #selectedEM := #statSelectedEMIdentRf;
	    #selectedUnit := #statSelectedUnitIdentRf;
	END_REGION
	
	
END_FUNCTION_BLOCK

FUNCTION "DemoIdentMv" : Void   // FC69, LAD
TITLE = Demo: IDENT_FC / Demo: Ident
AUTHOR : SICAR
FAMILY : Demo
VERSION : 1.0
// Demo fuer Anwendung Ident Bausteine / Demo for usage of ident moduls
// stored: IsIECCheckEnabled true, SetENOAutomatically true
   // Ret_Val : Ret_Val
BEGIN

REGION Network 1: Änderungshistorie / ChangeLog
   // Die Änderungshistorie wird nur in englischer Editiersprache geführt.
   // Change log table:
   // Version | Date | Expert in charge | Changes applied
   // -------|---------|-------------|--------------------------------------------
   // 05.00.00 | 01.09.2023 | SICAR | First released version
END_REGION

REGION Network 2: Call: Ident MV
   // Demonstrate the call and function of an optical reader MV device
END_REGION

REGION Network 3: Schreiben reader 1 / Define reading informations
   // Schreibe den String "Siemens" in die zu schreibende Datenstrucktur des RFID Geräts / Write the String "Siemens" in the writting structur of the FB
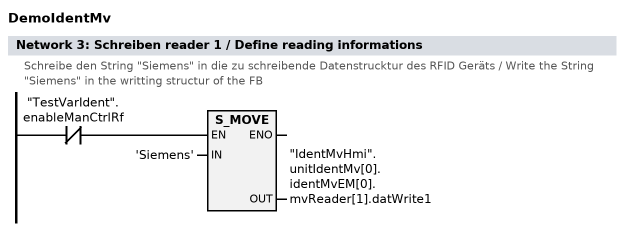
   RUNG wire#powerrail
      I_Contact( "TestVarIdent".enableManCtrlRf )
      S_Move(in := 'Siemens', out => "IdentMvHmi".unitIdentMv[0].identMvEM[0].mvReader[1].datWrite1)
   END_RUNG
   // the same network as SCL:
   IF NOT "TestVarIdent".enableManCtrlRf THEN
       "IdentMvHmi".unitIdentMv[0].identMvEM[0].mvReader[1].datWrite1 := 'Siemens';
   END_IF;
END_REGION
END_FUNCTION

FUNCTION_BLOCK "GetIdentMv"
{ S7_Optimized_Access := 'TRUE' ; Published := 'TRUE' }
VERSION : 0.1
   VAR_INPUT 
      identMvAllUnits { ExternalAccessible := 'False'; ExternalVisible := 'False'; ExternalWritable := 'False'} : Array[0.."NO_OF_UNITS"] of "typeEMIdentMv";   // HMI: motorstarter values
      numberOfMvReaders : USInt;
   END_VAR

   VAR_OUTPUT 
      selectedUnit : USInt;
      selectedEM : USInt;
      error : Word;
   END_VAR

   VAR_IN_OUT 
      IdentMvInterfaceHmi : "typeIdentMvHmi";
   END_VAR

   VAR 
      statSelectedEMIdentMv : USInt := 1;
      statSelectedUnitIdentRMv : USInt := 1;   // HMI: Selected unit
   END_VAR

   VAR_TEMP 
      tempEnable : Bool;   // Temporary value for input 'enable'
      tempMvReader : Array[0.."NO_OF_MV_IDENT_DEVICES"] of "LSicar_typeIdentInterfaceHmi";
      tempIndexIdentMv : USInt;
      tempNoOfidertMv : USInt;
   END_VAR

   VAR CONSTANT 
      "INVALID UNIT" : Word := 16#7001;   // non existant unit
      "INVALID EM" : Word := 16#7002;   // non existant em
      OK : Word := 16#7000;
   END_VAR


BEGIN
	REGION BLOCK INFO HEADER
	    //===============================================================================
	    // Siemens AG / (c)Copyright 2024
	    //-------------------------------------------------------------------------------
	    // Title:            LAF_GetMotorstarterSignals
	    // Comment/Function: This block reads diagnostic information of a Motorstarter depending
	    //                   on the unit and Control Module selected in the HMI by the user.
	    // Library/Family:   Automation Framework / Motorstarter Diagnostic
	    // Author:           Siemens Digital Industries
	    // Tested with:      S7-1517TF V3.1
	    // Engineering:      TIA Portal V19
	    // Restrictions:     
	    //                   Required UDTs: LAF_typeDriveDiagConfig, LAF_typeDriveDiagInterfaceHmi
	    // Requirements:     S7-1500(T), MC_Version V8.0
	    //-------------------------------------------------------------------------------
	    // Change log table:
	    // Version  | Date       | Expert in charge        | Changes applied
	    //----------|------------|-------------------------|-----------------------------
	    // 01.00.00 | 05.06.2024 | SIMATIC Systems Support | First released version
	    //===============================================================================
	END_REGION BLOCK INFO HEADER
	
	REGION DESCRIPTION
	(/*
	This block reads diagnostic information (control inputs and outputs) of a Motorstarter. 
	At runtime, this block is enabled when the ET200SP Motorstarter screen is shown in the HMI. 
	Based on the selected motorstarter object in the HMI by the user. The shown information in the HMI depends on the
	Unit and Cotrol Module selected. 
	*/)
	END_REGION DESCRIPTION
	
	REGION INPUTS
	    //working with static values to keep the last selected value when opening for the first time the screen  
	  
	    #statSelectedUnitIdentRMv := #IdentMvInterfaceHmi.selectedUnit;
	    #statSelectedEMIdentMv := #IdentMvInterfaceHmi.selectedEM;
	
	END_REGION INPUTS
	
	REGION ASSIGNING TEMPORARY VALUES
	    // Statement section REGION
	    IF #statSelectedUnitIdentRMv <= "NO_OF_UNITS" THEN
	        IF #statSelectedEMIdentMv < "NO_OF_EM" THEN
	            #tempMvReader := #identMvAllUnits[#statSelectedUnitIdentRMv].identMvEM[#statSelectedEMIdentMv].mvReader;
	            #tempNoOfidertMv := #numberOfMvReaders;
	            #error := #OK;
	        ELSE
	            #error := #"INVALID EM";
	        END_IF;
	
	    ELSE
	        #error := #"INVALID UNIT";
	    END_IF;
	
	
	END_REGION
	
	
	REGION OUTPUTS
	    // Statement section REGION
	    #IdentMvInterfaceHmi.mvReader := #tempMvReader;
	    #selectedEM := #statSelectedEMIdentMv;
	    #selectedUnit := #statSelectedUnitIdentRMv;
	END_REGION
	
	
END_FUNCTION_BLOCK

FUNCTION "SafetyState" : Void   // FC97, LAD
// stored: SetENOAutomatically false
   VAR CONSTANT
      TRUE : Bool := TRUE;
      FALSE : Bool;
   END_VAR
   VAR_TEMP   // added for the SCL form of the ladder/FBD networks
      _w1 : Bool;
   END_VAR
BEGIN

REGION Network 1: Stack Door Common Monitoring#1
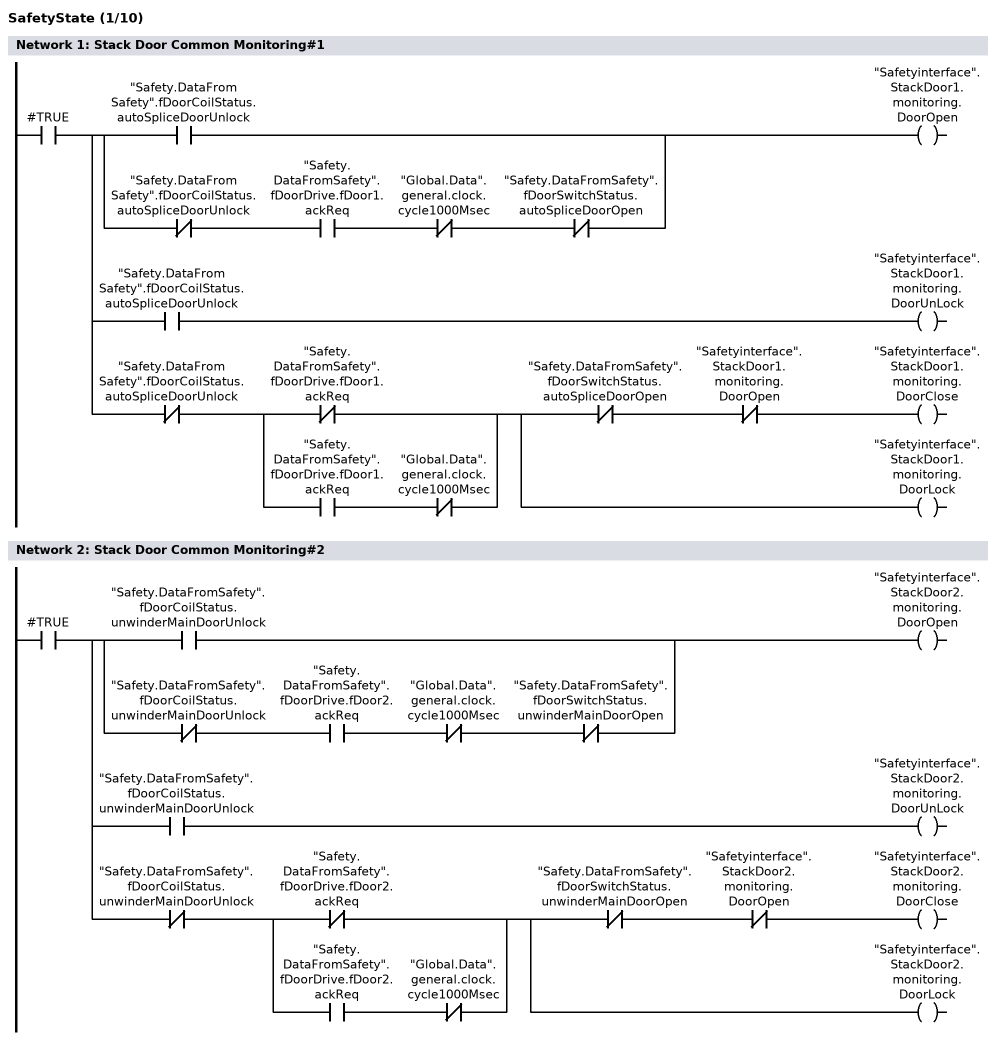
   RUNG wire#powerrail
      Contact( #TRUE )
      wire#w1
      Contact( "Safety.DataFromSafety".fDoorCoilStatus.autoSpliceDoorUnlock )
      wire#w2
      Coil( "Safetyinterface".StackDoor1.monitoring.DoorOpen )
   END_RUNG
   RUNG wire#w1
      I_Contact( "Safety.DataFromSafety".fDoorCoilStatus.autoSpliceDoorUnlock )
      Contact( "Safety.DataFromSafety".fDoorDrive.fDoor1.ackReq )
      I_Contact( "Global.Data".general.clock.cycle1000Msec )
      I_Contact( "Safety.DataFromSafety".fDoorSwitchStatus.autoSpliceDoorOpen )
   END_RUNG wire#w2
   RUNG wire#w1
      Contact( "Safety.DataFromSafety".fDoorCoilStatus.autoSpliceDoorUnlock )
      Coil( "Safetyinterface".StackDoor1.monitoring.DoorUnLock )
   END_RUNG
   RUNG wire#w1
      I_Contact( "Safety.DataFromSafety".fDoorCoilStatus.autoSpliceDoorUnlock )
      wire#w3
      I_Contact( "Safety.DataFromSafety".fDoorDrive.fDoor1.ackReq )
      wire#w4
      I_Contact( "Safety.DataFromSafety".fDoorSwitchStatus.autoSpliceDoorOpen )
      I_Contact( "Safetyinterface".StackDoor1.monitoring.DoorOpen )
      Coil( "Safetyinterface".StackDoor1.monitoring.DoorClose )
   END_RUNG
   RUNG wire#w3
      Contact( "Safety.DataFromSafety".fDoorDrive.fDoor1.ackReq )
      I_Contact( "Global.Data".general.clock.cycle1000Msec )
   END_RUNG wire#w4
   RUNG wire#w4
      Coil( "Safetyinterface".StackDoor1.monitoring.DoorLock )
   END_RUNG
   // the same network as SCL:
   "Safetyinterface".StackDoor1.monitoring.DoorOpen := #TRUE AND ("Safety.DataFromSafety".fDoorCoilStatus.autoSpliceDoorUnlock OR (NOT "Safety.DataFromSafety".fDoorCoilStatus.autoSpliceDoorUnlock AND "Safety.DataFromSafety".fDoorDrive.fDoor1.ackReq AND NOT "Global.Data".general.clock.cycle1000Msec AND NOT "Safety.DataFromSafety".fDoorSwitchStatus.autoSpliceDoorOpen));
   "Safetyinterface".StackDoor1.monitoring.DoorUnLock := #TRUE AND "Safety.DataFromSafety".fDoorCoilStatus.autoSpliceDoorUnlock;
   #_w1 := #TRUE AND NOT "Safety.DataFromSafety".fDoorCoilStatus.autoSpliceDoorUnlock AND (NOT "Safety.DataFromSafety".fDoorDrive.fDoor1.ackReq OR ("Safety.DataFromSafety".fDoorDrive.fDoor1.ackReq AND NOT "Global.Data".general.clock.cycle1000Msec));
   "Safetyinterface".StackDoor1.monitoring.DoorClose := #_w1 AND NOT "Safety.DataFromSafety".fDoorSwitchStatus.autoSpliceDoorOpen AND NOT "Safetyinterface".StackDoor1.monitoring.DoorOpen;
   "Safetyinterface".StackDoor1.monitoring.DoorLock := #_w1;
END_REGION

REGION Network 2: Stack Door Common Monitoring#2
   RUNG wire#powerrail
      Contact( #TRUE )
      wire#w1
      Contact( "Safety.DataFromSafety".fDoorCoilStatus.unwinderMainDoorUnlock )
      wire#w2
      Coil( "Safetyinterface".StackDoor2.monitoring.DoorOpen )
   END_RUNG
   RUNG wire#w1
      I_Contact( "Safety.DataFromSafety".fDoorCoilStatus.unwinderMainDoorUnlock )
      Contact( "Safety.DataFromSafety".fDoorDrive.fDoor2.ackReq )
      I_Contact( "Global.Data".general.clock.cycle1000Msec )
      I_Contact( "Safety.DataFromSafety".fDoorSwitchStatus.unwinderMainDoorOpen )
   END_RUNG wire#w2
   RUNG wire#w1
      Contact( "Safety.DataFromSafety".fDoorCoilStatus.unwinderMainDoorUnlock )
      Coil( "Safetyinterface".StackDoor2.monitoring.DoorUnLock )
   END_RUNG
   RUNG wire#w1
      I_Contact( "Safety.DataFromSafety".fDoorCoilStatus.unwinderMainDoorUnlock )
      wire#w3
      I_Contact( "Safety.DataFromSafety".fDoorDrive.fDoor2.ackReq )
      wire#w4
      I_Contact( "Safety.DataFromSafety".fDoorSwitchStatus.unwinderMainDoorOpen )
      I_Contact( "Safetyinterface".StackDoor2.monitoring.DoorOpen )
      Coil( "Safetyinterface".StackDoor2.monitoring.DoorClose )
   END_RUNG
   RUNG wire#w3
      Contact( "Safety.DataFromSafety".fDoorDrive.fDoor2.ackReq )
      I_Contact( "Global.Data".general.clock.cycle1000Msec )
   END_RUNG wire#w4
   RUNG wire#w4
      Coil( "Safetyinterface".StackDoor2.monitoring.DoorLock )
   END_RUNG
   // the same network as SCL:
   "Safetyinterface".StackDoor2.monitoring.DoorOpen := #TRUE AND ("Safety.DataFromSafety".fDoorCoilStatus.unwinderMainDoorUnlock OR (NOT "Safety.DataFromSafety".fDoorCoilStatus.unwinderMainDoorUnlock AND "Safety.DataFromSafety".fDoorDrive.fDoor2.ackReq AND NOT "Global.Data".general.clock.cycle1000Msec AND NOT "Safety.DataFromSafety".fDoorSwitchStatus.unwinderMainDoorOpen));
   "Safetyinterface".StackDoor2.monitoring.DoorUnLock := #TRUE AND "Safety.DataFromSafety".fDoorCoilStatus.unwinderMainDoorUnlock;
   #_w1 := #TRUE AND NOT "Safety.DataFromSafety".fDoorCoilStatus.unwinderMainDoorUnlock AND (NOT "Safety.DataFromSafety".fDoorDrive.fDoor2.ackReq OR ("Safety.DataFromSafety".fDoorDrive.fDoor2.ackReq AND NOT "Global.Data".general.clock.cycle1000Msec));
   "Safetyinterface".StackDoor2.monitoring.DoorClose := #_w1 AND NOT "Safety.DataFromSafety".fDoorSwitchStatus.unwinderMainDoorOpen AND NOT "Safetyinterface".StackDoor2.monitoring.DoorOpen;
   "Safetyinterface".StackDoor2.monitoring.DoorLock := #_w1;
END_REGION

REGION Network 3: Stack Door Common Monitoring#3
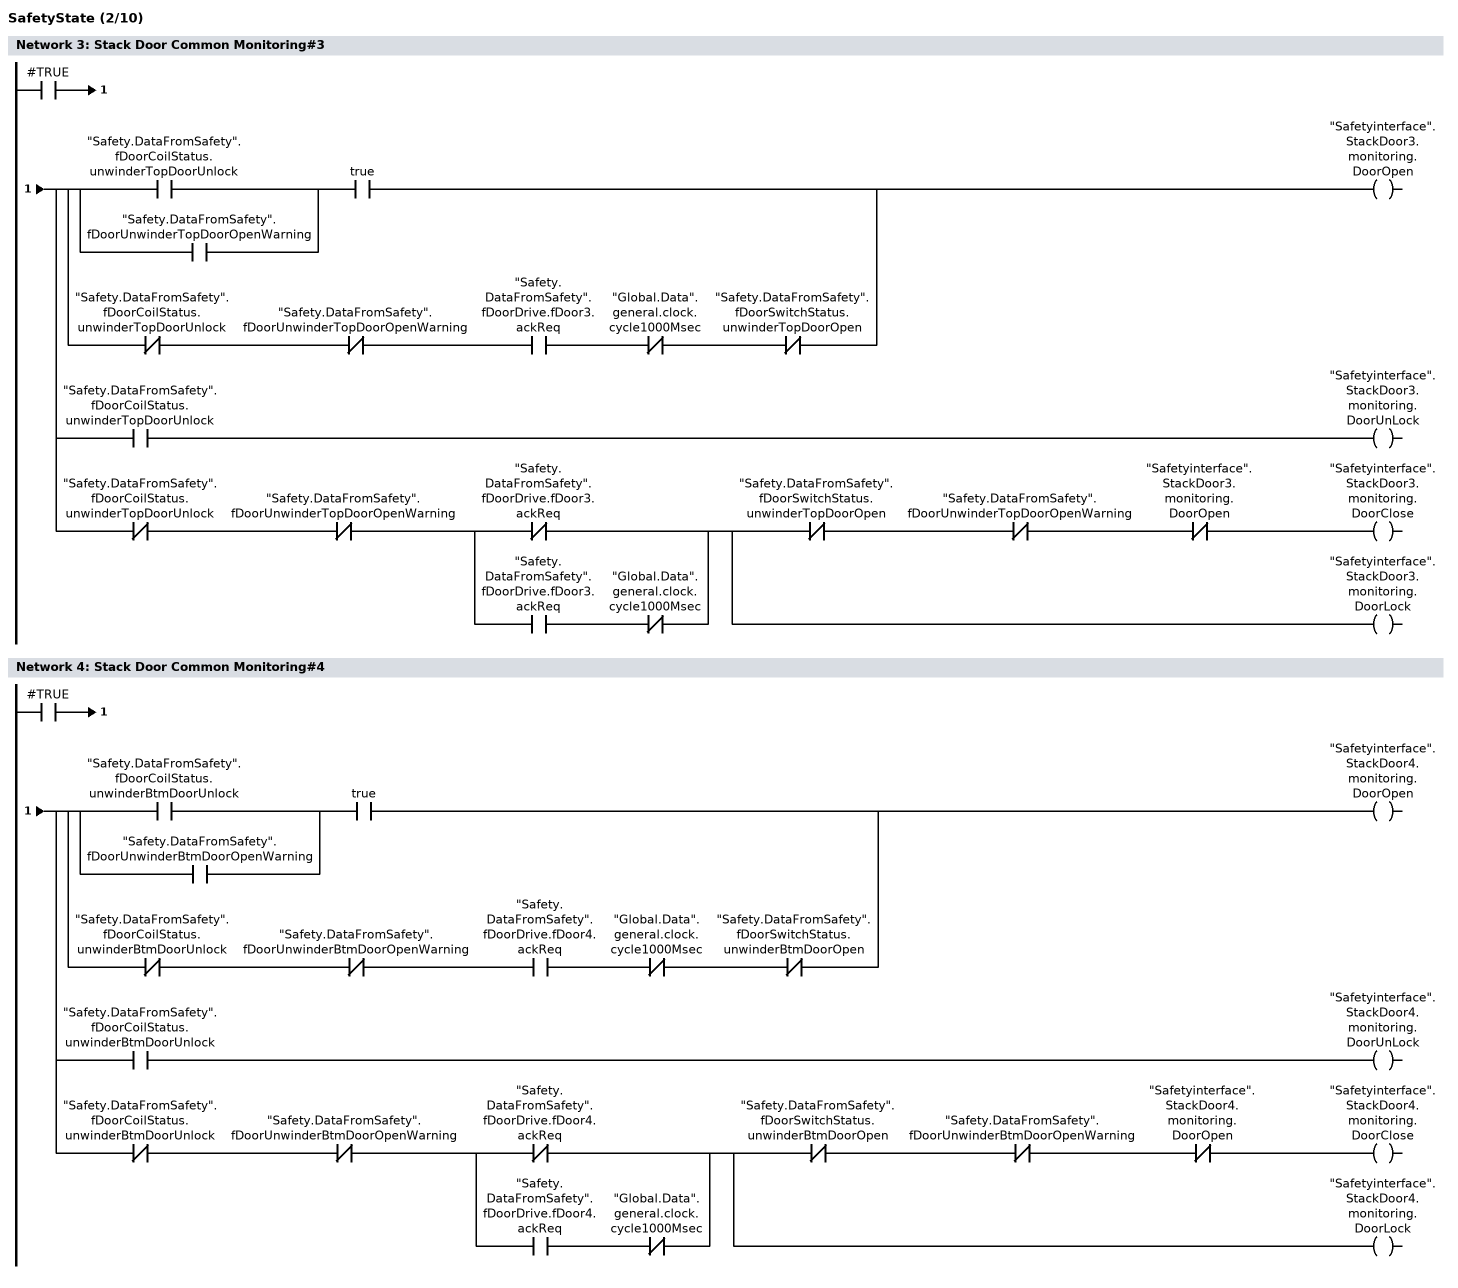
   RUNG wire#powerrail
      Contact( #TRUE )
      wire#w1
      Contact( "Safety.DataFromSafety".fDoorCoilStatus.unwinderTopDoorUnlock )
      wire#w2
      Contact( true )
      wire#w3
      Coil( "Safetyinterface".StackDoor3.monitoring.DoorOpen )
   END_RUNG
   RUNG wire#w1
      Contact( "Safety.DataFromSafety".fDoorUnwinderTopDoorOpenWarning )
   END_RUNG wire#w2
   RUNG wire#w1
      I_Contact( "Safety.DataFromSafety".fDoorCoilStatus.unwinderTopDoorUnlock )
      I_Contact( "Safety.DataFromSafety".fDoorUnwinderTopDoorOpenWarning )
      Contact( "Safety.DataFromSafety".fDoorDrive.fDoor3.ackReq )
      I_Contact( "Global.Data".general.clock.cycle1000Msec )
      I_Contact( "Safety.DataFromSafety".fDoorSwitchStatus.unwinderTopDoorOpen )
   END_RUNG wire#w3
   RUNG wire#w1
      Contact( "Safety.DataFromSafety".fDoorCoilStatus.unwinderTopDoorUnlock )
      Coil( "Safetyinterface".StackDoor3.monitoring.DoorUnLock )
   END_RUNG
   RUNG wire#w1
      I_Contact( "Safety.DataFromSafety".fDoorCoilStatus.unwinderTopDoorUnlock )
      I_Contact( "Safety.DataFromSafety".fDoorUnwinderTopDoorOpenWarning )
      wire#w4
      I_Contact( "Safety.DataFromSafety".fDoorDrive.fDoor3.ackReq )
      wire#w5
      I_Contact( "Safety.DataFromSafety".fDoorSwitchStatus.unwinderTopDoorOpen )
      I_Contact( "Safety.DataFromSafety".fDoorUnwinderTopDoorOpenWarning )
      I_Contact( "Safetyinterface".StackDoor3.monitoring.DoorOpen )
      Coil( "Safetyinterface".StackDoor3.monitoring.DoorClose )
   END_RUNG
   RUNG wire#w4
      Contact( "Safety.DataFromSafety".fDoorDrive.fDoor3.ackReq )
      I_Contact( "Global.Data".general.clock.cycle1000Msec )
   END_RUNG wire#w5
   RUNG wire#w5
      Coil( "Safetyinterface".StackDoor3.monitoring.DoorLock )
   END_RUNG
   // the same network as SCL:
   "Safetyinterface".StackDoor3.monitoring.DoorOpen := #TRUE AND ((("Safety.DataFromSafety".fDoorCoilStatus.unwinderTopDoorUnlock OR "Safety.DataFromSafety".fDoorUnwinderTopDoorOpenWarning) AND true) OR (NOT "Safety.DataFromSafety".fDoorCoilStatus.unwinderTopDoorUnlock AND NOT "Safety.DataFromSafety".fDoorUnwinderTopDoorOpenWarning AND "Safety.DataFromSafety".fDoorDrive.fDoor3.ackReq AND NOT "Global.Data".general.clock.cycle1000Msec AND NOT "Safety.DataFromSafety".fDoorSwitchStatus.unwinderTopDoorOpen));
   "Safetyinterface".StackDoor3.monitoring.DoorUnLock := #TRUE AND "Safety.DataFromSafety".fDoorCoilStatus.unwinderTopDoorUnlock;
   #_w1 := #TRUE AND NOT "Safety.DataFromSafety".fDoorCoilStatus.unwinderTopDoorUnlock AND NOT "Safety.DataFromSafety".fDoorUnwinderTopDoorOpenWarning AND (NOT "Safety.DataFromSafety".fDoorDrive.fDoor3.ackReq OR ("Safety.DataFromSafety".fDoorDrive.fDoor3.ackReq AND NOT "Global.Data".general.clock.cycle1000Msec));
   "Safetyinterface".StackDoor3.monitoring.DoorClose := #_w1 AND NOT "Safety.DataFromSafety".fDoorSwitchStatus.unwinderTopDoorOpen AND NOT "Safety.DataFromSafety".fDoorUnwinderTopDoorOpenWarning AND NOT "Safetyinterface".StackDoor3.monitoring.DoorOpen;
   "Safetyinterface".StackDoor3.monitoring.DoorLock := #_w1;
END_REGION

REGION Network 4: Stack Door Common Monitoring#4
   RUNG wire#powerrail
      Contact( #TRUE )
      wire#w1
      Contact( "Safety.DataFromSafety".fDoorCoilStatus.unwinderBtmDoorUnlock )
      wire#w2
      Contact( true )
      wire#w3
      Coil( "Safetyinterface".StackDoor4.monitoring.DoorOpen )
   END_RUNG
   RUNG wire#w1
      Contact( "Safety.DataFromSafety".fDoorUnwinderBtmDoorOpenWarning )
   END_RUNG wire#w2
   RUNG wire#w1
      I_Contact( "Safety.DataFromSafety".fDoorCoilStatus.unwinderBtmDoorUnlock )
      I_Contact( "Safety.DataFromSafety".fDoorUnwinderBtmDoorOpenWarning )
      Contact( "Safety.DataFromSafety".fDoorDrive.fDoor4.ackReq )
      I_Contact( "Global.Data".general.clock.cycle1000Msec )
      I_Contact( "Safety.DataFromSafety".fDoorSwitchStatus.unwinderBtmDoorOpen )
   END_RUNG wire#w3
   RUNG wire#w1
      Contact( "Safety.DataFromSafety".fDoorCoilStatus.unwinderBtmDoorUnlock )
      Coil( "Safetyinterface".StackDoor4.monitoring.DoorUnLock )
   END_RUNG
   RUNG wire#w1
      I_Contact( "Safety.DataFromSafety".fDoorCoilStatus.unwinderBtmDoorUnlock )
      I_Contact( "Safety.DataFromSafety".fDoorUnwinderBtmDoorOpenWarning )
      wire#w4
      I_Contact( "Safety.DataFromSafety".fDoorDrive.fDoor4.ackReq )
      wire#w5
      I_Contact( "Safety.DataFromSafety".fDoorSwitchStatus.unwinderBtmDoorOpen )
      I_Contact( "Safety.DataFromSafety".fDoorUnwinderBtmDoorOpenWarning )
      I_Contact( "Safetyinterface".StackDoor4.monitoring.DoorOpen )
      Coil( "Safetyinterface".StackDoor4.monitoring.DoorClose )
   END_RUNG
   RUNG wire#w4
      Contact( "Safety.DataFromSafety".fDoorDrive.fDoor4.ackReq )
      I_Contact( "Global.Data".general.clock.cycle1000Msec )
   END_RUNG wire#w5
   RUNG wire#w5
      Coil( "Safetyinterface".StackDoor4.monitoring.DoorLock )
   END_RUNG
   // the same network as SCL:
   "Safetyinterface".StackDoor4.monitoring.DoorOpen := #TRUE AND ((("Safety.DataFromSafety".fDoorCoilStatus.unwinderBtmDoorUnlock OR "Safety.DataFromSafety".fDoorUnwinderBtmDoorOpenWarning) AND true) OR (NOT "Safety.DataFromSafety".fDoorCoilStatus.unwinderBtmDoorUnlock AND NOT "Safety.DataFromSafety".fDoorUnwinderBtmDoorOpenWarning AND "Safety.DataFromSafety".fDoorDrive.fDoor4.ackReq AND NOT "Global.Data".general.clock.cycle1000Msec AND NOT "Safety.DataFromSafety".fDoorSwitchStatus.unwinderBtmDoorOpen));
   "Safetyinterface".StackDoor4.monitoring.DoorUnLock := #TRUE AND "Safety.DataFromSafety".fDoorCoilStatus.unwinderBtmDoorUnlock;
   #_w1 := #TRUE AND NOT "Safety.DataFromSafety".fDoorCoilStatus.unwinderBtmDoorUnlock AND NOT "Safety.DataFromSafety".fDoorUnwinderBtmDoorOpenWarning AND (NOT "Safety.DataFromSafety".fDoorDrive.fDoor4.ackReq OR ("Safety.DataFromSafety".fDoorDrive.fDoor4.ackReq AND NOT "Global.Data".general.clock.cycle1000Msec));
   "Safetyinterface".StackDoor4.monitoring.DoorClose := #_w1 AND NOT "Safety.DataFromSafety".fDoorSwitchStatus.unwinderBtmDoorOpen AND NOT "Safety.DataFromSafety".fDoorUnwinderBtmDoorOpenWarning AND NOT "Safetyinterface".StackDoor4.monitoring.DoorOpen;
   "Safetyinterface".StackDoor4.monitoring.DoorLock := #_w1;
END_REGION

REGION Network 5: Stack Door Common Command#5
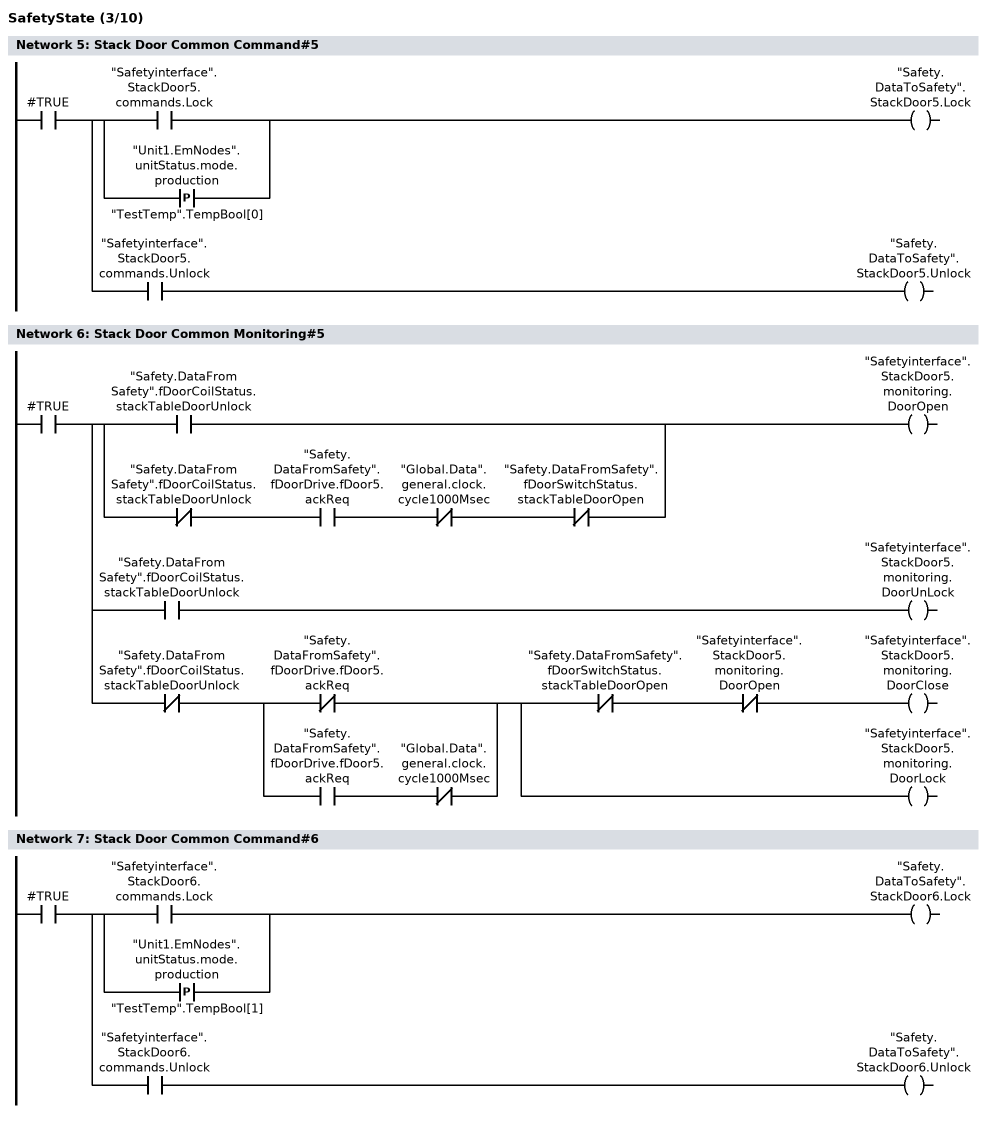
   RUNG wire#powerrail
      Contact( #TRUE )
      wire#w1
      Contact( "Safetyinterface".StackDoor5.commands.Lock )
      wire#w2
      Coil( "Safety.DataToSafety".StackDoor5.Lock )
   END_RUNG
   RUNG wire#w1
      P_Contact(operand := "Unit1.EmNodes".unitStatus.mode.production, bit := "TestTemp".TempBool[0])
   END_RUNG wire#w2
   RUNG wire#w1
      Contact( "Safetyinterface".StackDoor5.commands.Unlock )
      Coil( "Safety.DataToSafety".StackDoor5.Unlock )
   END_RUNG
   // the same network as SCL:
   #_w1 := #TRUE AND "Unit1.EmNodes".unitStatus.mode.production AND NOT "TestTemp".TempBool[0];   // rising edge of "Unit1.EmNodes".unitStatus.mode.production
   "TestTemp".TempBool[0] := "Unit1.EmNodes".unitStatus.mode.production;
   "Safety.DataToSafety".StackDoor5.Lock := (#TRUE AND "Safetyinterface".StackDoor5.commands.Lock) OR #_w1;
   "Safety.DataToSafety".StackDoor5.Unlock := #TRUE AND "Safetyinterface".StackDoor5.commands.Unlock;
END_REGION

REGION Network 6: Stack Door Common Monitoring#5
   RUNG wire#powerrail
      Contact( #TRUE )
      wire#w1
      Contact( "Safety.DataFromSafety".fDoorCoilStatus.stackTableDoorUnlock )
      wire#w2
      Coil( "Safetyinterface".StackDoor5.monitoring.DoorOpen )
   END_RUNG
   RUNG wire#w1
      I_Contact( "Safety.DataFromSafety".fDoorCoilStatus.stackTableDoorUnlock )
      Contact( "Safety.DataFromSafety".fDoorDrive.fDoor5.ackReq )
      I_Contact( "Global.Data".general.clock.cycle1000Msec )
      I_Contact( "Safety.DataFromSafety".fDoorSwitchStatus.stackTableDoorOpen )
   END_RUNG wire#w2
   RUNG wire#w1
      Contact( "Safety.DataFromSafety".fDoorCoilStatus.stackTableDoorUnlock )
      Coil( "Safetyinterface".StackDoor5.monitoring.DoorUnLock )
   END_RUNG
   RUNG wire#w1
      I_Contact( "Safety.DataFromSafety".fDoorCoilStatus.stackTableDoorUnlock )
      wire#w3
      I_Contact( "Safety.DataFromSafety".fDoorDrive.fDoor5.ackReq )
      wire#w4
      I_Contact( "Safety.DataFromSafety".fDoorSwitchStatus.stackTableDoorOpen )
      I_Contact( "Safetyinterface".StackDoor5.monitoring.DoorOpen )
      Coil( "Safetyinterface".StackDoor5.monitoring.DoorClose )
   END_RUNG
   RUNG wire#w3
      Contact( "Safety.DataFromSafety".fDoorDrive.fDoor5.ackReq )
      I_Contact( "Global.Data".general.clock.cycle1000Msec )
   END_RUNG wire#w4
   RUNG wire#w4
      Coil( "Safetyinterface".StackDoor5.monitoring.DoorLock )
   END_RUNG
   // the same network as SCL:
   "Safetyinterface".StackDoor5.monitoring.DoorOpen := #TRUE AND ("Safety.DataFromSafety".fDoorCoilStatus.stackTableDoorUnlock OR (NOT "Safety.DataFromSafety".fDoorCoilStatus.stackTableDoorUnlock AND "Safety.DataFromSafety".fDoorDrive.fDoor5.ackReq AND NOT "Global.Data".general.clock.cycle1000Msec AND NOT "Safety.DataFromSafety".fDoorSwitchStatus.stackTableDoorOpen));
   "Safetyinterface".StackDoor5.monitoring.DoorUnLock := #TRUE AND "Safety.DataFromSafety".fDoorCoilStatus.stackTableDoorUnlock;
   #_w1 := #TRUE AND NOT "Safety.DataFromSafety".fDoorCoilStatus.stackTableDoorUnlock AND (NOT "Safety.DataFromSafety".fDoorDrive.fDoor5.ackReq OR ("Safety.DataFromSafety".fDoorDrive.fDoor5.ackReq AND NOT "Global.Data".general.clock.cycle1000Msec));
   "Safetyinterface".StackDoor5.monitoring.DoorClose := #_w1 AND NOT "Safety.DataFromSafety".fDoorSwitchStatus.stackTableDoorOpen AND NOT "Safetyinterface".StackDoor5.monitoring.DoorOpen;
   "Safetyinterface".StackDoor5.monitoring.DoorLock := #_w1;
END_REGION

REGION Network 7: Stack Door Common Command#6
   RUNG wire#powerrail
      Contact( #TRUE )
      wire#w1
      Contact( "Safetyinterface".StackDoor6.commands.Lock )
      wire#w2
      Coil( "Safety.DataToSafety".StackDoor6.Lock )
   END_RUNG
   RUNG wire#w1
      P_Contact(operand := "Unit1.EmNodes".unitStatus.mode.production, bit := "TestTemp".TempBool[1])
   END_RUNG wire#w2
   RUNG wire#w1
      Contact( "Safetyinterface".StackDoor6.commands.Unlock )
      Coil( "Safety.DataToSafety".StackDoor6.Unlock )
   END_RUNG
   // the same network as SCL:
   #_w1 := #TRUE AND "Unit1.EmNodes".unitStatus.mode.production AND NOT "TestTemp".TempBool[1];   // rising edge of "Unit1.EmNodes".unitStatus.mode.production
   "TestTemp".TempBool[1] := "Unit1.EmNodes".unitStatus.mode.production;
   "Safety.DataToSafety".StackDoor6.Lock := (#TRUE AND "Safetyinterface".StackDoor6.commands.Lock) OR #_w1;
   "Safety.DataToSafety".StackDoor6.Unlock := #TRUE AND "Safetyinterface".StackDoor6.commands.Unlock;
END_REGION

REGION Network 8: Stack Door Common Monitoring#6
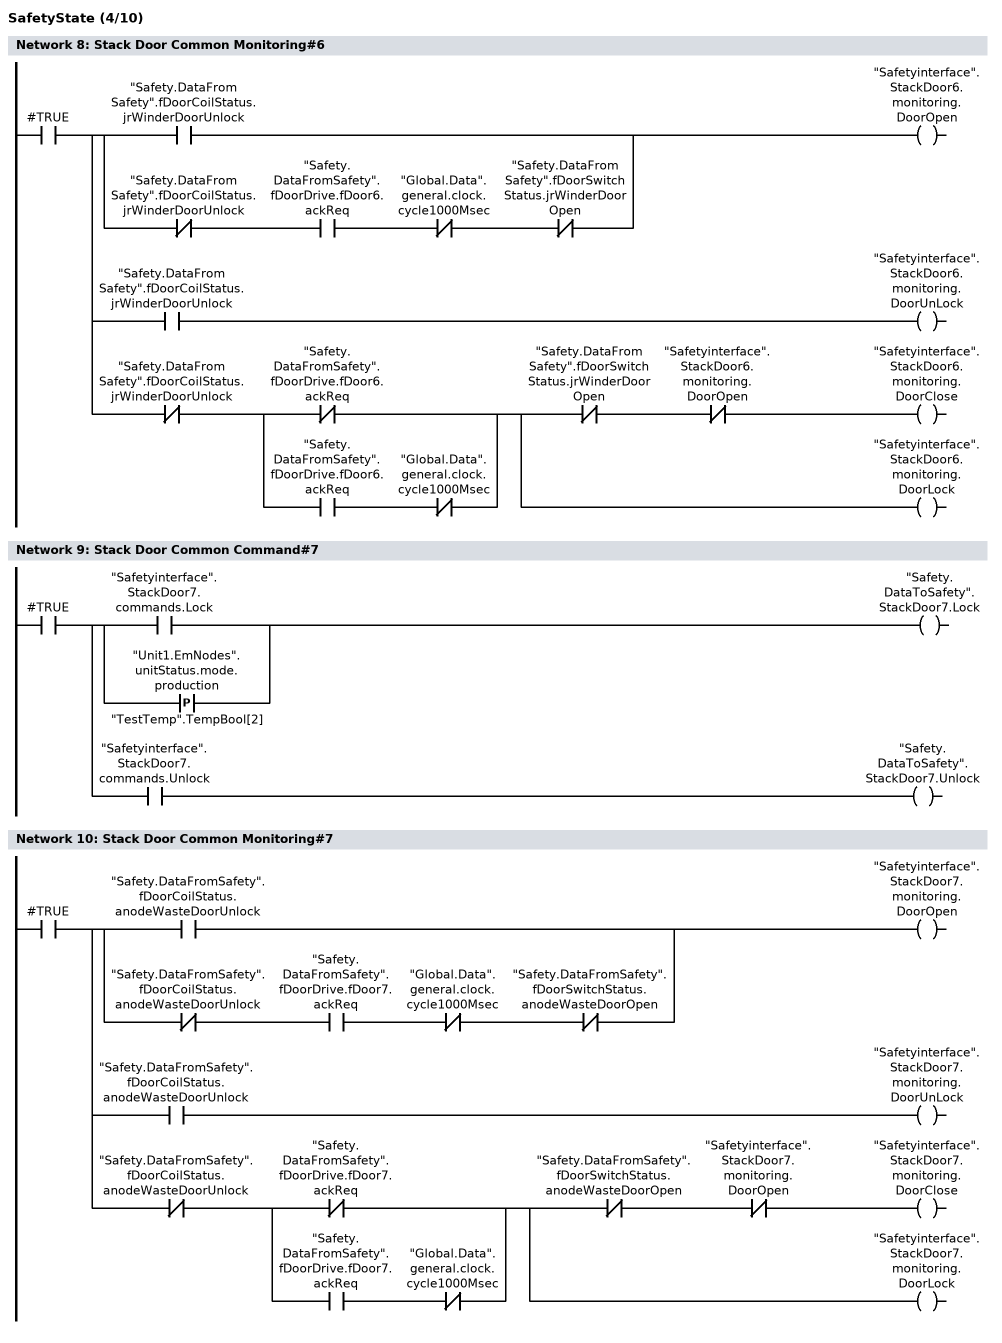
   RUNG wire#powerrail
      Contact( #TRUE )
      wire#w1
      Contact( "Safety.DataFromSafety".fDoorCoilStatus.jrWinderDoorUnlock )
      wire#w2
      Coil( "Safetyinterface".StackDoor6.monitoring.DoorOpen )
   END_RUNG
   RUNG wire#w1
      I_Contact( "Safety.DataFromSafety".fDoorCoilStatus.jrWinderDoorUnlock )
      Contact( "Safety.DataFromSafety".fDoorDrive.fDoor6.ackReq )
      I_Contact( "Global.Data".general.clock.cycle1000Msec )
      I_Contact( "Safety.DataFromSafety".fDoorSwitchStatus.jrWinderDoorOpen )
   END_RUNG wire#w2
   RUNG wire#w1
      Contact( "Safety.DataFromSafety".fDoorCoilStatus.jrWinderDoorUnlock )
      Coil( "Safetyinterface".StackDoor6.monitoring.DoorUnLock )
   END_RUNG
   RUNG wire#w1
      I_Contact( "Safety.DataFromSafety".fDoorCoilStatus.jrWinderDoorUnlock )
      wire#w3
      I_Contact( "Safety.DataFromSafety".fDoorDrive.fDoor6.ackReq )
      wire#w4
      I_Contact( "Safety.DataFromSafety".fDoorSwitchStatus.jrWinderDoorOpen )
      I_Contact( "Safetyinterface".StackDoor6.monitoring.DoorOpen )
      Coil( "Safetyinterface".StackDoor6.monitoring.DoorClose )
   END_RUNG
   RUNG wire#w3
      Contact( "Safety.DataFromSafety".fDoorDrive.fDoor6.ackReq )
      I_Contact( "Global.Data".general.clock.cycle1000Msec )
   END_RUNG wire#w4
   RUNG wire#w4
      Coil( "Safetyinterface".StackDoor6.monitoring.DoorLock )
   END_RUNG
   // the same network as SCL:
   "Safetyinterface".StackDoor6.monitoring.DoorOpen := #TRUE AND ("Safety.DataFromSafety".fDoorCoilStatus.jrWinderDoorUnlock OR (NOT "Safety.DataFromSafety".fDoorCoilStatus.jrWinderDoorUnlock AND "Safety.DataFromSafety".fDoorDrive.fDoor6.ackReq AND NOT "Global.Data".general.clock.cycle1000Msec AND NOT "Safety.DataFromSafety".fDoorSwitchStatus.jrWinderDoorOpen));
   "Safetyinterface".StackDoor6.monitoring.DoorUnLock := #TRUE AND "Safety.DataFromSafety".fDoorCoilStatus.jrWinderDoorUnlock;
   #_w1 := #TRUE AND NOT "Safety.DataFromSafety".fDoorCoilStatus.jrWinderDoorUnlock AND (NOT "Safety.DataFromSafety".fDoorDrive.fDoor6.ackReq OR ("Safety.DataFromSafety".fDoorDrive.fDoor6.ackReq AND NOT "Global.Data".general.clock.cycle1000Msec));
   "Safetyinterface".StackDoor6.monitoring.DoorClose := #_w1 AND NOT "Safety.DataFromSafety".fDoorSwitchStatus.jrWinderDoorOpen AND NOT "Safetyinterface".StackDoor6.monitoring.DoorOpen;
   "Safetyinterface".StackDoor6.monitoring.DoorLock := #_w1;
END_REGION

REGION Network 9: Stack Door Common Command#7
   RUNG wire#powerrail
      Contact( #TRUE )
      wire#w1
      Contact( "Safetyinterface".StackDoor7.commands.Lock )
      wire#w2
      Coil( "Safety.DataToSafety".StackDoor7.Lock )
   END_RUNG
   RUNG wire#w1
      P_Contact(operand := "Unit1.EmNodes".unitStatus.mode.production, bit := "TestTemp".TempBool[2])
   END_RUNG wire#w2
   RUNG wire#w1
      Contact( "Safetyinterface".StackDoor7.commands.Unlock )
      Coil( "Safety.DataToSafety".StackDoor7.Unlock )
   END_RUNG
   // the same network as SCL:
   #_w1 := #TRUE AND "Unit1.EmNodes".unitStatus.mode.production AND NOT "TestTemp".TempBool[2];   // rising edge of "Unit1.EmNodes".unitStatus.mode.production
   "TestTemp".TempBool[2] := "Unit1.EmNodes".unitStatus.mode.production;
   "Safety.DataToSafety".StackDoor7.Lock := (#TRUE AND "Safetyinterface".StackDoor7.commands.Lock) OR #_w1;
   "Safety.DataToSafety".StackDoor7.Unlock := #TRUE AND "Safetyinterface".StackDoor7.commands.Unlock;
END_REGION

